(* Stop button *)
	xTmp:=	NOT(T_Visu.T_CtrleAction.xExecute);
	xTmpTeach:=((T_Visu.T_PlcParam.dwActualPage = 310) OR (T_Visu.T_PlcParam.dwActualPage = 410)) AND (bButtonPanelLocked = 16#10);
	IF xTmp THEN
		RisingEdgeStopButton(CLK:=xStopButton);
		IF RisingEdgeStopButton.Q AND ((bButtonPanelLocked = 16#0) OR xTmpTeach) THEN
		(* pane locked *)
			bButtonPanelLocked:=16#20;
			(* activ stop process *)
			T_Visu.T_CtrleAction.xExecute:=TRUE;
			CASE T_Visu.T_PlcParam.dwActualPage OF
			10:	T_Visu.T_CtrleAction.iFunction:=800;
			20:	T_Visu.T_CtrleAction.iFunction:=800;
			30:	T_Visu.T_CtrleAction.iFunction:=800;
			110:	T_Visu.T_CtrleAction.iFunction:=800;
				T_Visu.ptrT_ExchgParam^.T_Visu.T_Message.iState:=121;
			210:	T_Visu.T_CtrleAction.iFunction:=301;
				T_Visu.ptrT_ExchgParam^.T_Visu.T_Message.iState:=121;
			220:	T_Visu.T_CtrleAction.iFunction:=403;
				T_Visu.ptrT_ExchgParam^.T_Visu.T_Message.iState:=121;
			310:	T_Visu.T_CtrleAction.iFunction:=301;
				T_Visu.ptrT_ExchgParam^.T_Visu.T_Message.iState:=121;
			330:	T_Visu.T_CtrleAction.iFunction:=800;
				T_Visu.ptrT_ExchgParam^.T_Visu.T_Message.iState:=121;
			410:	T_Visu.T_CtrleAction.iFunction:=301;
				T_Visu.ptrT_ExchgParam^.T_Visu.T_Message.iState:=121;
			ELSE
				T_Visu.T_CtrleAction.xExecute:=FALSE;
			END_CASE
		END_IF
		(* manage falling edge stop button *)
		FallingEdgeStopButton(CLK:=xStopButton AND T_ConfigPage.xMaskBtStop);
		IF FallingEdgeStopButton.Q AND (bButtonPanelLocked AND 16#20) = 16#20 THEN
			bButtonPanelLocked:=bButtonPanelLocked XOR 16#20; END_IF
	ELSE
		RisingEdgeStopButton(CLK:=FALSE);
		FallingEdgeStopButton(CLK:=TRUE);
	END_IF
END_ACTION
ACTION CtrlTaskBar:
(* Management Bt navigation panel *)
	RisingEdgeTouchScreenNavPanel(CLK:=	T_Visu.ptrT_ExchgParam^.T_TouchScreenNavPanel.wActivBt <> 0);
	FallingEdgeTouchScreenNavPanel(CLK:=T_Visu.ptrT_ExchgParam^.T_TouchScreenNavPanel.wActivBt <> 0);
	xTmp:=	NOT(xChangePage)
			AND T_Visu.T_CtrleAction.xDone
			AND NOT(T_Visu.T_CtrleAction.xExecute)
			AND NOT(T_StartUp.T_State.xBlockChangeMovementVisu)
			AND NOT(T_StartUp.T_State.xBlockVisuNavigation)
			AND ((T_Visu.ptrT_ExchgParam^. T_TouchScreenNavPanel.wNotMasktext AND T_Visu.ptrT_ExchgParam^.T_TouchScreenNavPanel.wActivBt) <> 0);
	IF xTmp THEN
		(* activ action of rising edge *)
		IF RisingEdgeTouchScreenNavPanel.Q THEN
			ii:=1;
			wTmp:=T_Visu.ptrT_ExchgParam^.T_TouchScreenNavPanel.wActivBt;
			WHILE wTmp <> 16#0 DO
				IF (wTmp AND 16#1) = 16#1 THEN EXIT; END_IF
				wTmp:=ROR(wTmp,1);
				ii:=ii+1;
			END_WHILE
			T_Visu.T_CtrleAction.iFunction:=T_ConfigPage.aiFTrigActionTouchScreenNavPanel[ii];
			CASE T_Visu.ptrT_ExchgParam^.T_Visu.bActivSpecialLayer OF
				0: 	wNormalLayerActivTask:=T_Visu.ptrT_ExchgParam^.T_TouchScreenNavPanel.wActivBt;
					wNormalLayerActivPage:=T_Visu.T_CtrleAction.iFunction - 10000;
					T_Visu.ptrT_ExchgParam^.T_TouchScreenNavPanel.wState:=wNormalLayerActivTask;
					wTmpNormalLayerActivTask:=ii;
				1:	wSpecialLayerGeneralActivTask:=T_Visu.ptrT_ExchgParam^.T_TouchScreenNavPanel.wActivBt;
					wSpecialLayerGeneralActivPage:=T_Visu.T_CtrleAction.iFunction - 10000;
					T_Visu.ptrT_ExchgParam^.T_TouchScreenNavPanel.wState:=wSpecialLayerGeneralActivTask;
					wTmpSpecialLayerGeneralActivTask:=ii;
				2:	wSpecialLayerToolRotActivTask:=T_Visu.ptrT_ExchgParam^.T_TouchScreenNavPanel.wActivBt;
					wSpecialLayerToolRotActivPage:=T_Visu.T_CtrleAction.iFunction - 10000;
					T_Visu.ptrT_ExchgParam^.T_TouchScreenNavPanel.wState:=wSpecialLayerToolRotActivTask;
					wTmpSpecialLayerToolRotActivTask:=ii;
				3:	wSpecialLayerWireFeedActivTask:=T_Visu.ptrT_ExchgParam^.T_TouchScreenNavPanel.wActivBt;
					wSpecialLayerWireFeedActivPage:=T_Visu.T_CtrleAction.iFunction - 10000;
					T_Visu.ptrT_ExchgParam^.T_TouchScreenNavPanel.wState:=wSpecialLayerWireFeedActivTask;
					wTmpSpecialLayerWireFeedActivTask:=ii;
				4:	wSpecialLayerGrindAxisActivTask:=T_Visu.ptrT_ExchgParam^.T_TouchScreenNavPanel.wActivBt;
					wSpecialLayerGrindAxisActivPage:=T_Visu.T_CtrleAction.iFunction - 10000;
					T_Visu.ptrT_ExchgParam^.T_TouchScreenNavPanel.wState:=wSpecialLayerGrindAxisActivTask;
					wTmpSpecialLayerGrindAxisActivTask:=ii;
			END_CASE;
			IF ((INT_TO_WORD(T_Visu.ptrT_ExchgParam^.T_TouchScreenBtPanel.iStateBtLeft) AND 16#10) = 16#10) THEN
				T_Visu.T_CtrleAction.iFunction:=3;
				xResetParaListValue:=TRUE;
			END_IF;
			T_Visu.ptrT_ExchgParam^.T_TouchScreenNavPanel.wActivBt:=0;
			T_Visu.T_CtrleAction.xExecute:=TRUE;
		END_IF;
	ELSE
		T_Visu.ptrT_ExchgParam^.T_TouchScreenNavPanel.wActivBt:=0;
	END_IF;
(*22.12.2009: KFS 	{	*)
(* Management BT Tool  (additionel external buttons) only for MicroRod *)
	IF xMicroRodActive THEN
		(* ToolTension button *)
		xTmp:=	NOT(xChangePage) AND T_Visu.T_CtrleAction.xDone AND
				NOT(T_Visu.T_CtrleAction.xExecute) 	AND T_Visu.T_CtrleProcess.xDone AND (bStateMachine <>2);
		IF xTmp THEN
(*03.03.2017: KFS { *)
			RisingEdgeBtToolTension(CLK:=xToolTensionButton);
			IF RisingEdgeBtToolTension.Q THEN
				IF  T_Visu.ptrT_ExchgParam^.T_Cylinder.xToolTension AND	T_Visu.ptrT_ExchgParam^.T_Cylinder.xCylToolLeft AND T_Visu.ptrT_ExchgParam^.T_Cylinder.xCylToolRight	THEN
					T_Visu.T_CtrleAction.iFunction:=510;
					T_Visu.T_CtrleAction.xExecute:=TRUE;
				END_IF;
				IF  NOT (T_Visu.ptrT_ExchgParam^.T_Cylinder.xToolTension) THEN
					T_Visu.T_CtrleAction.iFunction:=510;
					T_Visu.T_CtrleAction.xExecute:=TRUE;
				END_IF;
			END_IF;
			RisingEdgeBtToolLeft(CLK:=xToolLeftButton);
			IF RisingEdgeBtToolLeft.Q THEN
				IF NOT T_Visu.ptrT_ExchgParam^.T_Cylinder.xToolTension  THEN
					T_Visu.T_CtrleAction.iFunction:=511;
					T_Visu.T_CtrleAction.xExecute:=TRUE;
				END_IF;
				IF  T_Visu.ptrT_ExchgParam^.T_Cylinder.xToolTension  AND NOT(T_Visu.ptrT_ExchgParam^.T_Cylinder.xCylToolLeft) THEN
					T_Visu.T_CtrleAction.iFunction:=511;
					T_Visu.T_CtrleAction.xExecute:=TRUE;
				END_IF;
			END_IF;
			RisingEdgeBtToolRight(CLK:=xToolRightButton);
			IF RisingEdgeBtToolRight.Q THEN
				IF NOT T_Visu.ptrT_ExchgParam^.T_Cylinder.xToolTension  THEN
					T_Visu.T_CtrleAction.iFunction:=512;
					T_Visu.T_CtrleAction.xExecute:=TRUE;
				END_IF;
				IF  T_Visu.ptrT_ExchgParam^.T_Cylinder.xToolTension  AND NOT(T_Visu.ptrT_ExchgParam^.T_Cylinder.xCylToolRight) THEN
					T_Visu.T_CtrleAction.iFunction:=512;
					T_Visu.T_CtrleAction.xExecute:=TRUE;
				END_IF;
			END_IF;
(*03.03.2017: KFS } *)
			RisingEdgeBtToolCenter(CLK:=xToolCenterButton);
			IF RisingEdgeBtToolCenter.Q THEN
				T_Visu.T_CtrleAction.iFunction:=513;
				T_Visu.T_CtrleAction.xExecute:=TRUE;
			END_IF;
			RisingEdgeBtToolPrismaLeft(CLK:=xToolPrismaLeftButton);
			IF RisingEdgeBtToolPrismaLeft.Q THEN
				T_Visu.T_CtrleAction.iFunction:=514;
				T_Visu.T_CtrleAction.xExecute:=TRUE;
			END_IF;
			RisingEdgeBtToolPrismaRight(CLK:=xToolPrismaRightButton);
			IF RisingEdgeBtToolPrismaRight.Q THEN
				T_Visu.T_CtrleAction.iFunction:=515;
				T_Visu.T_CtrleAction.xExecute:=TRUE;
			END_IF;
		ELSE
			IF   NOT(T_Visu.T_CtrleAction.xExecute) AND T_Visu.T_CtrleAction.xDone  THEN
				RisingEdgeBtToolTension(CLK:=FALSE);
				RisingEdgeBtToolLeft(CLK:=FALSE);
				RisingEdgeBtToolRight(CLK:=FALSE);
				RisingEdgeBtToolCenter(CLK:=FALSE);
				RisingEdgeBtToolPrismaLeft(CLK:=FALSE);
				RisingEdgeBtToolPrismaRight(CLK:=FALSE);
			END_IF;
		END_IF;
	END_IF;
(*22.12.2009: KFS 	}	*)
END_ACTION
ACTION CtrlVisuFunction:
(************************************************************************************************************************************************************************)
(***************                                          start of the management for call a function of the visualisation interface                                           ********************)
(************************************************************************************************************************************************************************)
(* waiting for executing action *)
	(* ...monitor Key panel "Enter" *)
	RisingEdgeKeyPanel_Enter(CLK:=T_Visu.ptrT_ExchgParam^.T_Visu.xKey_Enter);
	(* ...monitor Key panel "Esc" *)
	RisingEdgeKeyPanel_Esc(CLK:=T_Visu.ptrT_ExchgParam^.T_Visu.xKey_Escape);
	IF RisingEdgeKeyPanel_Esc.Q THEN tTimeOutAction:=TimerAction.ET; END_IF
	(*... not ready *)
	TimerNotReady(IN:=FALSE, PT:=T#2s);
	T_Visu.T_CtrleAction.xNotReady:=TimerNotReady.Q;

(* ...message *)
	RisingEdgeActionNotReady(CLK:=T_Visu.T_CtrleAction.xNotReady);
	IF RisingEdgeActionNotReady.Q AND T_Visu.ptrT_ExchgParam^.T_Visu.T_Message.iState < 200 THEN
		T_Visu.ptrT_ExchgParam^.T_Visu.T_Message.iState:=101; END_IF
	(* Release 'Not ready' action control structure *)
	FallingEdgeActionNotReady(CLK:=T_Visu.T_CtrleAction.xNotReady);
	IF FallingEdgeActionNotReady.Q THEN
		IF (T_Visu.ptrT_ExchgParam^.T_Visu.T_Message.iState =101) THEN
			T_Visu.ptrT_ExchgParam^.T_Visu.T_Message.iState:=0;
		END_IF;
		T_Visu.T_CtrleAction.xExecute:=FALSE;
		T_Visu.T_CtrleAction.xDone:=TRUE;
		T_Visu.T_CtrleAction.xErr:=FALSE;
		T_Visu.T_CtrleAction.udiErrorID:=0;
		iStepAction:=1;
		(*
		iStepActionRef:=1;
		iStepActionNovRam:=1;
		*)
		xStepActionDone:=FALSE;
		TimerAction(IN:=FALSE);
	END_IF
	(* ...done *)
	RisingEdgeActionDone(CLK:=T_Visu.T_CtrleAction.xDone);
	IF RisingEdgeActionDone.Q THEN
		(* disable mask stop action *)
		(*wStopActionMaskBtPanelRight:=16#0;*)
		(*xWaitingReleaseStopBtPanel:=FALSE;*)
		IF T_Visu.T_CtrleAction.iFunction > 100
		    AND (T_Visu.ptrT_ExchgParam^.T_Visu.T_Message.iState = 0 OR (T_Visu.ptrT_ExchgParam^.T_Visu.T_Message.iState  > 100 AND T_Visu.ptrT_ExchgParam^.T_Visu.T_Message.iState < 200)) THEN
			IF NOT TimerAction.Q AND NOT FallingEdgeActionNotReady.Q THEN
				IF NOT(xBlockConfirmMessage) THEN
					(* call confirmation message *)
					T_Visu.ptrT_ExchgParam^.T_Visu.T_Message.iState
						:=iFctReturnConfMessage(iNumAction:=T_Visu.T_CtrleAction.iFunction);
				ELSE
					xBlockConfirmMessage:=FALSE;
				END_IF;
			(* call cancelled message *)
			ELSE T_Visu.ptrT_ExchgParam^.T_Visu.T_Message.iState:=5; END_IF
		END_IF
	END_IF
	(* ...error *)
	RisingEdgeActionError(CLK:=T_Visu.T_CtrleAction.xErr);
	IF RisingEdgeActionError.Q THEN
	(* call function bloc action error *)
		(*fbQvisError(	udiActionError:=T_Visu.T_CtrleAction.udiErrorID,
					T_Message:=T_Visu.ptrT_ExchgParam^.T_Visu.T_Message);*)
		(* Init. variable *)
		T_Visu.T_CtrleAction.xExecute:=FALSE;
		T_Visu.T_CtrleAction.xDone:=TRUE;
		T_Visu.T_CtrleAction.xErr:=FALSE;
		T_Visu.T_CtrleAction.xNotReady:=FALSE;
		T_Visu.T_CtrleAction.udiErrorID:=0;
		iStepAction:=1;
		(*
		iStepActionRef:=1;
		iStepActionNovRam:=1;
		*)
		xStepActionDone:=FALSE;
	END_IF
	(* ...reset *)
	RisingEdgeResetAction(CLK:=T_Visu.T_CtrleAction.xReset);
	IF RisingEdgeResetAction.Q THEN
		(* Init. variable *)
		T_Visu.T_CtrleAction.xExecute:=FALSE;
		T_Visu.T_CtrleAction.xDone:=TRUE;
		T_Visu.T_CtrleAction.xErr:=FALSE;
		T_Visu.T_CtrleAction.xNotReady:=FALSE;
		T_Visu.T_CtrleAction.udiErrorID:=0;
		iStepAction:=1;
		(*
		iStepActionRef:=1;
		iStepActionNovRam:=1;
		*)
		xStepActionDone:=FALSE;
		TimerAction(IN:=FALSE);
		(* Release reset *)
		T_Visu.T_CtrleAction.xReset:=FALSE;
	END_IF

	(* Execute Function *)
	RisingEdgeExecuteAction(CLK:=T_Visu.T_CtrleAction.xExecute);
	IF RisingEdgeExecuteAction.Q THEN
		(* confirm action execution *)
		T_Visu.T_CtrleAction.xExecute:=FALSE;
		CASE T_Visu.T_CtrleAction.iFunction OF
			(* Set parameter page *)
			3:	xSetParameterPage:=TRUE;
				tTimeOutAction:=T#3s;
			(* Change Page Button Panel Left *)
			6:	xBtPanelLeftChangePage:=TRUE;
				tTimeOutAction:=T#3s;
	(*SOA 13.01.2023  { *)
			(* Change Page Button Panel Right *)
			7:	xBtPanelRightChangePage:=TRUE;
				tTimeOutAction:=T#3s;
	(*SOA 13.01.2023  } *)
			(* next page vertical *)
			12:	xNextPageVertical:=TRUE;
				tTimeOutAction:=T#3s;
			(* Delete error List *)
			20:	xDeleteErrorList:=TRUE;
				tTimeOutAction:=T#3s;
			(* Reset error *)
			99:	xResetError:=TRUE;
				tTimeOutAction:=T#3s;
			(* Open Overlay for input measured tool diameter *)
			101:	xOverlayMeasureToolDia:=TRUE;
				tTimeOutAction:=T#9999s;
			(* Plunge On/Off *)
			102:	xPlungeActivation:=TRUE;
				tTimeOutAction:=T#3s;
			(* Displace On/Off *)
			103:	xDisplaceActivation:=TRUE;
				tTimeOutAction:=T#3s;
			(* AutoGroove-->Block GrindFeeder On/Off *)
			104:	xBlockGrindFeederActivation:=TRUE;
				tTimeOutAction:=T#3s;
			(* AutoGroove-->ToolFeeder move to StartPos *)
			105:	xToolFeederMoveStartPos:=TRUE;
				tTimeOutAction:=T#3s;
			(* AutoGeometry and AutoGroove-->Switch On/Off all Axis Power *)
			106:	xToggleAllAxisPower:=TRUE;
				tTimeOutAction:=T#3s;
			(* AutoGeometry and AutoGroove-->ToolFeeder move to LoadPos *)
			107:	xToolFeederMoveLoadPos:=TRUE;
				tTimeOutAction:=T#3s;
(*08.07.2014: KFS	{	*)
			(* AutoGeometry -->WarmUp On/OFF *)
			108:	xWarmUp:=TRUE;
				tTimeOutAction:=T#3s;
(*08.07.2014: KFS	}	*)
			(* Correction Tool Diameter + *)
			110:	xCorrectionToolDiameterAdd:=TRUE;
				tTimeOutAction:=T#3s;
			(* Correction Tool Diameter ++ *)
			111:	xCorrectionToolDiameterAddMore:=TRUE;
				tTimeOutAction:=T#3s;
			(* Correction Tool Diameter - *)
			112:	xCorrectionToolDiameterSub:=TRUE;
				tTimeOutAction:=T#3s;
			(* Correction Tool Diameter -- *)
			113:	xCorrectionToolDiameterSubMore:=TRUE;
				tTimeOutAction:=T#3s;
			(* Reset Tool Diameter Correction *)
			114:	xResetToolDiameterCorrection:=TRUE;
				tTimeOutAction:=T#3s;
			(* Keypad Activation *)
			115: xKeyPadActivation:=TRUE;
				tTimeOutAction:=T#3s;
			(* Function Correction Tool Diameter *)
			116:	xFctCorrectionToolDiameter:=TRUE;
				tTimeOutAction:=T#3s;
			(* Select Prisma 1 or 2 Input *)
			120:	xSelectPrisma:=TRUE;
				tTimeOutAction:=T#3s;
			(* Set calculated ToolRotation Torque *)
			130:	xSetCalculToolRotTorque:=TRUE;
				tTimeOutAction:=T#3s;
			(* Reset calculated ToolRotation Torque *)
			131:	xResetCalculToolRotTorque:=TRUE;
				tTimeOutAction:=T#3s;
			(* Open Overlay for input the correction of the position of the GrindFeeder *)
			132:	xOverlayGrindFeedSetPlung:=TRUE;
				tTimeOutAction:=T#9999s;
	(*SOA 13.01.2023  { *)
			173:	xConfirmStartWarmUp:=TRUE;
				tTimeOutAction:=T#3s;
			(* Stop Warmupl  *)
			175: 	xStopWarmup:=TRUE;
				tTimeOutAction:=T#3s;
	(*SOA 13.01.2023  } *)
			(* Activation Section 1 *) (*
			201: (* 13.10.2010 KFS 	{ 	*)
				(*	xActivationSection1:=TRUE;
					tTimeOutAction:=T#3s;			*)
				(* 13.10.2010 KFS   }	 *) *)
			(* Activation Section 2 *)
			202:	xActivationSection2:=TRUE;
				tTimeOutAction:=T#3s;
			(* Activation Section 3 *)
			203:	xActivationSection3:=TRUE;
				tTimeOutAction:=T#3s;
			(* Activation Section 4 *)
			204:	xActivationSection4:=TRUE;
				tTimeOutAction:=T#3s;
			(* Set pitch equal *)
			205:	xSetPitchEqual:=TRUE;
				tTimeOutAction:=T#3s;
	(* 13.10.2022 SOA*)
			(* Activation Section 5 *)
			206:	xActivationSection5:=TRUE;
				tTimeOutAction:=T#3s;
			(* Activation Section 6 *)
			207:	xActivationSection6:=TRUE;
				tTimeOutAction:=T#3s;
	(* 13.10.2022 SOA*)
			(* TeachIN page *)
			301..399:	(* set pointer, default pointer axis slide *)
					ptrTeachINAxis:=ADR(T_Station.THardware.TAxisToolLeft);
					iSelectedAxis:=1;
					IF (T_Visu.T_PlcParam.dwActualPage = 210) THEN
						xSlowFast:=T_Visu.ptrT_ExchgParam^.T_TeachIn.xSlowFastToolRotation;
						CASE T_Visu.ptrT_ExchgParam^.T_TeachIn.iSelectAxisToolRotation OF
						1:	iSelectedAxis:=1;
							TParaAxisTeachIN:=T_Visu.ptrT_ExchgParam^.T_TeachIn.TParam_ToolLeft:=T_NovRam.T_Data.T_Standard.T_TeachINToolLeft;
							ptrTeachINAxis:=ADR(T_Station.THardware.TAxisToolLeft);
						2:	iSelectedAxis:=2;
							TParaAxisTeachIN:=T_Visu.ptrT_ExchgParam^.T_TeachIn.TParam_ToolCenter:=T_NovRam.T_Data.T_Standard.T_TeachINToolCenter;
							ptrTeachINAxis:=ADR(T_Station.THardware.TAxisToolCenter);
						3:	iSelectedAxis:=3;
							TParaAxisTeachIN:=T_Visu.ptrT_ExchgParam^.T_TeachIn.TParam_ToolRight:=T_NovRam.T_Data.T_Standard.T_TeachINToolRight;
							ptrTeachINAxis:=ADR(T_Station.THardware.TAxisToolRight);
						END_CASE
					END_IF;
					IF (T_Visu.T_PlcParam.dwActualPage = 30) OR (T_Visu.T_PlcParam.dwActualPage = 310) OR (T_Visu.T_PlcParam.dwActualPage = 320) OR (T_Visu.T_PlcParam.dwActualPage = 330) THEN
						iSelectedAxis:=4;
						xSlowFast:=T_Visu.ptrT_ExchgParam^.T_TeachIn.xSlowFastToolFeed;
						TParaAxisTeachIN:=T_Visu.ptrT_ExchgParam^.T_TeachIn.TParam_ToolFeeder:=T_NovRam.T_Data.T_Standard.T_TeachINToolFeeder;
						ptrTeachINAxis:=ADR(T_Station.THardware.TAxisToolFeeder);
					END_IF;
					IF (T_Visu.T_PlcParam.dwActualPage = 410) THEN
						xSlowFast:=T_Visu.ptrT_ExchgParam^.T_TeachIn.xSlowFastGrindFeeder;
						CASE T_Visu.ptrT_ExchgParam^.T_TeachIn.iSelectAxisGrind OF
						1:	iSelectedAxis:=5;
							TParaAxisTeachIN:=T_Visu.ptrT_ExchgParam^.T_TeachIn.TParam_GrindFeeder:=T_NovRam.T_Data.T_Standard.T_TeachINGrindFeeder;
							ptrTeachINAxis:=ADR(T_Station.THardware.TAxisGrindFeeder);
						2:	iSelectedAxis:=6;
							ptrTeachINAxis:=ADR(T_Station.THardware.TAxisGrindSpindle);
						END_CASE
					END_IF;
					CASE T_Visu.T_CtrleAction.iFunction OF
					(* Stop axis movement *)
					301:	xStopAxis:=TRUE;
						tTimeOutAction:=T#4s;
					(* Move Axis Absolut *)
					305:	IF (iSelectedAxis = 4) THEN
							IF xMicroRodActive THEN
								IF (T_Visu.ptrT_ExchgParam^.T_TeachIn.iSaveToolFeederPos = 0) THEN
									ptrTeachINAxis^.T_CtrleSingle.lrPosition:=T_Visu.ptrT_ExchgParam^.T_StationCommon.rNewToolFeederPosition;
								END_IF;
								IF (T_Visu.ptrT_ExchgParam^.T_TeachIn.iSaveToolFeederPos = 1) THEN
									ptrTeachINAxis^.T_CtrleSingle.lrPosition:=T_NovRam.T_Data.T_ProcessImageData.T_ProcessPara.rStartPosToolFeedAuto;
								END_IF;
								IF (T_Visu.ptrT_ExchgParam^.T_TeachIn.iSaveToolFeederPos = 2) THEN
									ptrTeachINAxis^.T_CtrleSingle.lrPosition:=T_NovRam.T_Data.T_ProcessImageData.T_CalibrationPara.rStartPosToolFeedCalib;
								END_IF;
								IF (T_Visu.ptrT_ExchgParam^.T_TeachIn.iSaveToolFeederPos = 3) THEN
									ptrTeachINAxis^.T_CtrleSingle.lrPosition:=T_NovRam.T_Data.T_ProcessImageData.T_CalibrationPara.rMeasurePosToolFeedCalib;
								END_IF;
								IF (T_Visu.ptrT_ExchgParam^.T_TeachIn.iSaveToolFeederPos = 4) THEN
									ptrTeachINAxis^.T_CtrleSingle.lrPosition:=T_NovRam.T_Data.T_Standard.T_AxisPosition.rLoadPosToolFeedAuto;
								END_IF;
								ptrTeachINAxis^.T_CtrleSingle.lrVelocity:=TParaAxisTeachIN.rPositionSpeed;
								xMoveAbsPosition:=TRUE;
							END_IF;
							IF NOT(xMicroRodActive) THEN
								ptrTeachINAxis^.T_CtrleSingle.lrDistance:=T_Visu.ptrT_ExchgParam^.T_StationCommon.rNewToolFeederPosition;
								ptrTeachINAxis^.T_CtrleSingle.lrVelocity:=TParaAxisTeachIN.rPositionSpeed;
								xMoveRelPosition:=TRUE;
							END_IF;
						END_IF;
						IF (iSelectedAxis = 5) THEN
							IF (T_Visu.ptrT_ExchgParam^.T_TeachIn.iSaveGrindFeederPos = 0) THEN
								ptrTeachINAxis^.T_CtrleSingle.lrPosition:=T_Visu.ptrT_ExchgParam^.T_StationCommon.rNewGrindFeederPosition;
							END_IF;
							IF (T_Visu.ptrT_ExchgParam^.T_TeachIn.iSaveGrindFeederPos = 1) THEN
								ptrTeachINAxis^.T_CtrleSingle.lrPosition:=T_NovRam.T_Data.T_ProcessImageData.T_ProcessPara.rToolDiameterProcess;
							END_IF;
							IF (T_Visu.ptrT_ExchgParam^.T_TeachIn.iSaveGrindFeederPos = 2) THEN
								ptrTeachINAxis^.T_CtrleSingle.lrPosition:=	T_NovRam.T_Data.T_ProcessImageData.T_ProcessPara.rToolDiameterProcess +
																	T_NovRam.T_Data.T_ProcessImageData.T_ProcessPara.rSecurityPosGrindFeedProcess;
							END_IF;
							IF (T_Visu.ptrT_ExchgParam^.T_TeachIn.iSaveGrindFeederPos = 3) THEN
								ptrTeachINAxis^.T_CtrleSingle.lrPosition:=T_NovRam.T_Data.T_ProcessImageData.T_PrismPara.rToolDiameterMin;;
							END_IF;
							IF (T_Visu.ptrT_ExchgParam^.T_TeachIn.iSaveGrindFeederPos = 4) THEN
								ptrTeachINAxis^.T_CtrleSingle.lrPosition:=T_NovRam.T_Data.T_ProcessImageData.T_PrismPara.rToolDiameterMax + T_NovRam.T_Data.T_Standard.T_TeachINGrindFeeder.rOffsetSWPosEndSwitch;
							END_IF;
							ptrTeachINAxis^.T_CtrleSingle.lrVelocity:=TParaAxisTeachIN.rPositionSpeed;
							xMoveAbsPosition:=TRUE;
						END_IF;
						tTimeOutAction:=T#999s;
					(* Move Inc Slow/Fast Pos *)
					310..311: IF NOT(xSlowFast) THEN
								ptrTeachINAxis^.T_CtrleSingle.lrDistance:=TParaAxisTeachIN.rIncSlow;
								ptrTeachINAxis^.T_CtrleSingle.lrVelocity:=TParaAxisTeachIN.rVelSlow;
							ELSE
								ptrTeachINAxis^.T_CtrleSingle.lrDistance:=TParaAxisTeachIN.rIncFast;
								ptrTeachINAxis^.T_CtrleSingle.lrVelocity:=TParaAxisTeachIN.rVelFast;
							END_IF
							xMoveRelPosition:=TRUE;
							tTimeOutAction:=T#200s;
					(* Move Inc Slow/Fast Neg *)
					312..313:	IF NOT(xSlowFast) THEN
								ptrTeachINAxis^.T_CtrleSingle.lrDistance:=TParaAxisTeachIN.rIncSlow * -1.0;
								ptrTeachINAxis^.T_CtrleSingle.lrVelocity:=TParaAxisTeachIN.rVelSlow;
							ELSE
								ptrTeachINAxis^.T_CtrleSingle.lrDistance:=TParaAxisTeachIN.rIncFast * -1.0;
								ptrTeachINAxis^.T_CtrleSingle.lrVelocity:=TParaAxisTeachIN.rVelFast;
							END_IF
							xMoveRelPosition:=TRUE;
							tTimeOutAction:=T#200s;
					(* Move Vel Slow/Fast Pos *)
					314..315:	IF NOT(xSlowFast) THEN
								ptrTeachINAxis^.T_CtrleSingle.lrVelocity:=TParaAxisTeachIN.rVelSlow;
							ELSE
								ptrTeachINAxis^.T_CtrleSingle.lrVelocity:=TParaAxisTeachIN.rVelFast;
							END_IF
							xMoveContinousVel:=TRUE;
							tTimeOutAction:=T#200s;
					(* Move Vel Slow/Fast Neg *)
					316..317:	IF NOT(xSlowFast) THEN
								ptrTeachINAxis^.T_CtrleSingle.lrVelocity:=TParaAxisTeachIN.rVelSlow * -1.0;
							ELSE
								ptrTeachINAxis^.T_CtrleSingle.lrVelocity:=TParaAxisTeachIN.rVelFast * -1.0;
							END_IF
							xMoveContinousVel:=TRUE;
							tTimeOutAction:=T#200s;
					(* Move Continuos Velocity *)
					318:		CASE iSelectedAxis OF
							1,2,3:	ptrTeachINAxis^.T_CtrleSingle.lrVelocity:=T_Visu.ptrT_ExchgParam^.T_StationCommon.rNewToolRotationSpeed;
							6:		ptrTeachINAxis^.T_CtrleSingle.lrVelocity:=T_Visu.ptrT_ExchgParam^.T_StationCommon.rNewGrindSpindleSpeed;
							END_CASE
							xMoveContinousVel:=TRUE;
							tTimeOutAction:=T#200s;
					(* Switch WireFeed Jog Speed Slow/Fast *)
					320:		IF ((iSelectedAxis = 1) OR (iSelectedAxis = 2) OR (iSelectedAxis = 3)) AND (T_Visu.T_PlcParam.dwActualPage <> 30) THEN
								xSlowFastJogToolRotation:=TRUE;
							END_IF;
							IF (iSelectedAxis = 4) OR (T_Visu.T_PlcParam.dwActualPage = 30) THEN
								xSlowFastJogToolFeeder:=TRUE;
							END_IF;
							IF (iSelectedAxis = 5) AND (T_Visu.T_PlcParam.dwActualPage <> 30) THEN
								xSlowFastJogGrindFeeder:=TRUE;
							END_IF;
							tTimeOutAction:=T#3s;
					(* Switch ToolRotation Master Slave *)
					321:		IF xMicroRodActive THEN
								(* ToolCenter --> Slave of ToolLeft only by MicroRod *)
								T_Station.THardware.TAxisToolCenter.T_CtrleSingle.lrGearDivider:=INT_TO_LREAL(T_Station.T_WorkTool.iBaseGearDivider);
								T_Station.THardware.TAxisToolCenter.T_CtrleSingle.lrGearFactor:=(	INT_TO_LREAL(T_Station.T_WorkTool.iBaseGearDivider) /
																								(T_Station.THardware.TAxisToolLeft.T_CtrleSingle.lrGearRatio /
																								T_Station.THardware.TAxisToolCenter.T_CtrleSingle.lrGearRatio)) * -1.0;

								(* ToolRight --> Slave of ToolLeft by MicroWire or Slave of ToolRight by MicroRod *)
								T_Station.THardware.TAxisToolRight.T_CtrleSingle.lrGearDivider:=INT_TO_LREAL(T_Station.T_WorkTool.iBaseGearDivider);
								T_Station.THardware.TAxisToolRight.T_CtrleSingle.lrGearFactor:=	INT_TO_LREAL(T_Station.T_WorkTool.iBaseGearDivider) /
																								(T_Station.THardware.TAxisToolLeft.T_CtrleSingle.lrGearRatio /
																								T_Station.THardware.TAxisToolRight.T_CtrleSingle.lrGearRatio);
							END_IF;
							IF NOT(xMicroRodActive) THEN
								(* ToolRight --> Slave of ToolRight by MicroWire *)
								T_Station.THardware.TAxisToolFeeder.T_CtrleSingle.lrGearDivider:=INT_TO_LREAL(T_Station.T_WorkTool.iBaseGearDivider);
								T_Station.THardware.TAxisToolFeeder.T_CtrleSingle.lrGearFactor:=	(INT_TO_LREAL(T_Station.T_WorkTool.iBaseGearDivider) /
																							(T_Station.THardware.TAxisToolFeeder.T_CtrleSingle.lrGearRatio /
																							T_Station.THardware.TAxisToolRight.T_CtrleSingle.lrGearRatio)) * -1.0;

								(* ToolRight --> Slave of ToolLeft by MicroWire or Slave of ToolRight by MicroRod *)
								T_Station.THardware.TAxisToolRight.T_CtrleSingle.lrGearDivider:=INT_TO_LREAL(T_Station.T_WorkTool.iBaseGearDivider);
								T_Station.THardware.TAxisToolRight.T_CtrleSingle.lrGearFactor:=	(INT_TO_LREAL(T_Station.T_WorkTool.iBaseGearDivider) /
																								(T_Station.THardware.TAxisToolLeft.T_CtrleSingle.lrGearRatio /
																								T_Station.THardware.TAxisToolRight.T_CtrleSingle.lrGearRatio)) * -1.0;
							END_IF;
							xSwitchMasterSlave:=TRUE;
							tTimeOutAction:=T#3s;
					(* Power axis *)
					322:		xToggleAxisPower:=TRUE;
							tTimeOutAction:=T#3s;
					(* Reset axis *)
					323:		xResetAxis:=TRUE;
							tTimeOutAction:=T#3s;
					(* Reference axis *)
					324:		xReferenceAxis:=TRUE;
							tTimeOutAction:=T#200s;
					(* Teach axis Position *)
					325:		xTeachPosition:=TRUE;
							tTimeOutAction:=T#6s;
					(* Calculate the position between the RefIndex and the RefSensor *)
					326:		xCalcAngleRefIndex:=TRUE;
							tTimeOutAction:=T#200s;

					(* CW /CCW *)
					330:		xCWCCW:=TRUE;
							tTimeOutAction:=T#3s;
					(* CylBrake *)
					331:		xCylBrake:=TRUE;
							tTimeOutAction:=T#3s;
					END_CASE;
			(* Station Function *)
			401..499:	xActivateStationFunction:=TRUE;
					iTmpStationFunctionNr:=T_Visu.T_CtrleAction.iFunction - 400;	(* Select Function Number 1 - 99 *)
					IF (iTmpStationFunctionNr = 20) THEN tTimeOutAction:=T#200s; ELSE tTimeOutAction:=T#3s;END_IF;
			(* Cylinder Function *)
			501..599:	(* set pointer, default pointer CylToolTension *)
					(* 1=CylToolTension, 2=CylToolLeftActive, 3=CylToolRightActive, 4=CylToolCenter,5=CylToolPrismaLeftActive, 6=CylToolPrismaRightActive *)
					ptrCylAction:=ADR(T_Station.THardware.TCylToolTension);
					iSelectedCylinder:=1;
					IF (T_Visu.T_PlcParam.dwActualPage = 230) THEN
						IF (T_Visu.ptrT_ExchgParam^.T_Cylinder.iSelectCylinder_Sonder1 = 1) THEN
							ptrCylAction:=ADR(T_Station.THardware.TCylToolTension);
							iSelectedCylinder:=1;
						ELSIF (T_Visu.ptrT_ExchgParam^.T_Cylinder.iSelectCylinder_Sonder1 = 2) THEN
							ptrCylAction:=ADR(T_Station.THardware.TCylToolLeftActive);
							iSelectedCylinder:=2;
						ELSIF (T_Visu.ptrT_ExchgParam^.T_Cylinder.iSelectCylinder_Sonder1 = 3) THEN
							ptrCylAction:=ADR(T_Station.THardware.TCylToolRightActive);
							iSelectedCylinder:=3;
						ELSIF (T_Visu.ptrT_ExchgParam^.T_Cylinder.iSelectCylinder_Sonder1 = 4) THEN
							ptrCylAction:=ADR(T_Station.THardware.TCylToolCenterActive);
							iSelectedCylinder:=4;
						ELSIF (T_Visu.ptrT_ExchgParam^.T_Cylinder.iSelectCylinder_Sonder1 = 5) THEN
							ptrCylAction:=ADR(T_Station.THardware.TCylToolPrismaLeftActive);
							iSelectedCylinder:=5;
						ELSIF (T_Visu.ptrT_ExchgParam^.T_Cylinder.iSelectCylinder_Sonder1 = 6) THEN
							ptrCylAction:=ADR(T_Station.THardware.TCylToolPrismaRightActive);
							iSelectedCylinder:=6;
						ELSE
							ptrCylAction:=ADR(T_Station.THardware.TCylToolTension);
							iSelectedCylinder:=1;
						END_IF;
					END_IF;
					(*Set pointer -->selection by the extern buttons*)
					IF (T_Visu.T_CtrleAction.iFunction = 510) THEN ptrCylAction:=ADR(T_Station.THardware.TCylToolTension);iSelectedCylinder:=1; END_IF;
					IF (T_Visu.T_CtrleAction.iFunction = 511) THEN ptrCylAction:=ADR(T_Station.THardware.TCylToolLeftActive);iSelectedCylinder:=2; END_IF;
					IF (T_Visu.T_CtrleAction.iFunction = 512) THEN ptrCylAction:=ADR(T_Station.THardware.TCylToolRightActive);iSelectedCylinder:=3; END_IF;
					IF (T_Visu.T_CtrleAction.iFunction = 513) THEN ptrCylAction:=ADR(T_Station.THardware.TCylToolCenterActive);iSelectedCylinder:=4; END_IF;
					IF (T_Visu.T_CtrleAction.iFunction = 514) THEN ptrCylAction:=ADR(T_Station.THardware.TCylToolPrismaLeftActive);iSelectedCylinder:=5; END_IF;
					IF (T_Visu.T_CtrleAction.iFunction = 515) THEN ptrCylAction:=ADR(T_Station.THardware.TCylToolPrismaRightActive);iSelectedCylinder:=6; END_IF;
					IF ((T_Visu.T_CtrleAction.iFunction >= 510) AND (T_Visu.T_CtrleAction.iFunction <= 515)) THEN
						T_Visu.T_CtrleAction.iFunction:=501;
					 END_IF;
					CASE T_Visu.T_CtrleAction.iFunction OF
					501:		xToggleCylinderState:=TRUE;
							IF ( iSelectedCylinder = 1) THEN
								IF (T_Visu.T_PlcParam.dwActualPage = 220) THEN
									ptrCylAction^.T_CtrleCyl.T_AnalogCylinder.rForceIn:=T_Visu.ptrT_ExchgParam^.T_InfoValueCommon.rToolTensionForce;
								ELSE
									IF (T_Visu.ptrT_ExchgParam^.T_Cylinder.iSelectToolTensionForce < 2) THEN
										(* Process work force *)
										ptrCylAction^.T_CtrleCyl.T_AnalogCylinder.rForceIn:=T_NovRam.T_Data.T_ProcessImageData.T_ProcessPara.rToolTensionProcess;
									END_IF;
									IF (T_Visu.ptrT_ExchgParam^.T_Cylinder.iSelectToolTensionForce > 1) THEN
										(* Setup (Cylinder Force) Force *)
										ptrCylAction^.T_CtrleCyl.T_AnalogCylinder.rForceIn:=T_NovRam.T_Data.T_Standard.T_Cyl_ToolTension.rForce;
									END_IF;
								END_IF;
							END_IF;
							tTimeOutAction:=T#2s;
					(* ToolTens force + *)
					502:		xToolTensForceAdd:=TRUE;
							tTimeOutAction:=T#2s;
					(* ToolTens force ++ *)
					503:		xToolTensForceAddMore:=TRUE;
							tTimeOutAction:=T#2s;
					(* ToolTens force - *)
					504:		xToolTensForceSub:=TRUE;
							tTimeOutAction:=T#2s;
					(* ToolTens force -- *)
					505:		xToolTensForceSubMore:=TRUE;
							tTimeOutAction:=T#2s;
					(* DO NOT USE FUNCTION 510,511,512,513,514,515 *)
					END_CASE;
			(* All process station *)
			601..699:	T_Process.iFunctNr:=T_Visu.T_CtrleAction.iFunction - 600;
					xActionProcStation:=TRUE;
					tTimeOutAction:=T#2s;
			(* All process machine *)
			701..799:	T_Process.iFunctNr:=T_Visu.T_CtrleAction.iFunction - 700;
					xActionProcMachine:=TRUE;
					(* Ref timeout 120s *)
					IF T_Visu.T_CtrleAction.iFunction = 710 THEN  tTimeOutAction:=T#120s; ELSE tTimeOutAction:=T#0.5s; END_IF
			(* Stop process *)
			800:		xStopProcess:=TRUE;
					tTimeOutAction:=T#30s;
			(* Stop cycle *)
			801:		xAction_StopCycle:=TRUE;
					tTimeOutAction:=T#30s;
			(* Copy profile to process value *)
			1001:	xAction_CopyProfileToProcess:=TRUE;
					tTimeOutAction:=T#10s;
			(* Load profile to process image *)
			1002:	xAction_LoadProfileToProcessImage:=TRUE;
					tTimeOutAction:=T#5s;
			(* Save profile to File *)
			1003:	xAction_SaveProfileToFile:=TRUE;
					tTimeOutAction:=T#5s;
			(* Delete Profile *)
			1004:	xActionDeleteProfile:=TRUE;
					tTimeOutAction:=T#5s;
			(* Save NovRAM with confirmation *)
			1005:	xAction_SaveNovRAM:=TRUE;
					tTimeOutAction:=T#6s;
			(* Save NovRAM without confirmation *)
			1006:	xAction_SaveNovRAMWithoutConfirm:=TRUE;
					tTimeOutAction:=T#10s;
			(* change page *)
			10001..10999:	xNavPanelChangePage:=TRUE;
						tTimeOutAction:=T#3s;
		END_CASE;
		(* Init. variable *)
		T_Visu.T_CtrleAction.xDone:=FALSE;
		T_Visu.T_CtrleAction.xNotReady:=FALSE;
		T_Visu.T_CtrleAction.xErr:=FALSE;
		T_Visu.T_CtrleAction.udiErrorID:=0;
		iStepAction:=1;
		iStepActionNovRam:=1;
		xStepActionDone:=FALSE;
		IF tTimeOutAction <> T#0s THEN TimerAction(IN:=FALSE); END_IF
		(* exit FB *)
		RETURN;
	END_IF;

(* Timer action *)
	IF tTimeOutAction <> T#0s THEN TimerAction(IN:=TRUE,PT:=tTimeOutAction); END_IF
	RisingEdgeTimeOut(CLK:=TimerAction.Q);
	IF RisingEdgeTimeOut.Q AND NOT(T_Visu.T_CtrleAction.xDone) AND NOT(T_Visu.T_CtrleAction.xErr) THEN
	(* Timeout action activ *)
		T_Visu.T_CtrleAction.xExecute:=FALSE;
		T_Visu.T_CtrleAction.xDone:=TRUE;
		T_Visu.T_CtrleAction.xNotReady:=FALSE;
		T_Visu.T_CtrleAction.xErr:=FALSE;
		T_Visu.T_CtrleAction.udiErrorID:=16#0;
		(* call confirmation message *)
		T_Visu.ptrT_ExchgParam^.T_Visu.T_Message.iState:=102;
(*			:=iFctReturnConfMessage(iNumAction:=-1);*)
		(* exit FB, do not continue the execution of action! *)
		RETURN;
	END_IF
(************************************************************************************************************************************************************************)
(***************                                          end  of the management for call a function of the visualisation interface                                           ********************)
(************************************************************************************************************************************************************************)
END_ACTION
ACTION MaskFunctionButton:
CASE T_Visu.T_PlcParam.dwActualPage OF
410:	CASE T_Visu.ptrT_ExchgParam^.T_TeachIn.iSelectAxisGrind OF
	1:	wForceMaskFunctionPanel:=16#2B;
		aiForceRTrigActionFunctionPanel[1]:=322;		(* On/Off *)
		aiForceRTrigActionFunctionPanel[2]:=323;		(* Reset *)
		aiForceRTrigActionFunctionPanel[3]:=0;
		aiForceRTrigActionFunctionPanel[4]:=320;		(* Slow / Fast *)
		aiForceRTrigActionFunctionPanel[5]:=0;
		aiForceRTrigActionFunctionPanel[6]:=325;		(* Save position *)
	2:	wForceMaskFunctionPanel:=16#2B;
		aiForceRTrigActionFunctionPanel[1]:=322;		(* On/Off *)
		aiForceRTrigActionFunctionPanel[2]:=323;		(* Reset *)
		aiForceRTrigActionFunctionPanel[3]:=0;
		aiForceRTrigActionFunctionPanel[4]:=330;		(* CW / CCW *)
		aiForceRTrigActionFunctionPanel[5]:=0;
		aiForceRTrigActionFunctionPanel[6]:=331;		(* CylBrake *)
	END_CASE
END_CASE
END_ACTION
ACTION Monitor_ActuatorState:
(* Monitoring Axis value *)
	(* ToolLeft Monitoring *)
	IF T_Station.THardware.TAxisToolLeft.T_CtrleSingle.xPower THEN
		T_Visu.ptrT_ExchgParam^.T_StationCommon.bStateAxisReelLeft:=T_Visu.ptrT_ExchgParam^.T_StationCommon.bStateAxisReelLeft OR 16#1;
	ELSE
		T_Visu.ptrT_ExchgParam^.T_StationCommon.bStateAxisReelLeft:=T_Visu.ptrT_ExchgParam^.T_StationCommon.bStateAxisReelLeft AND 16#FE;
	END_IF;
	IF NOT(T_Station.THardware.TAxisToolLeft.T_CtrleSingle.xNotMoving) THEN
		T_Visu.ptrT_ExchgParam^.T_StationCommon.bStateAxisReelLeft:=T_Visu.ptrT_ExchgParam^.T_StationCommon.bStateAxisReelLeft OR 16#2;
	ELSE
		T_Visu.ptrT_ExchgParam^.T_StationCommon.bStateAxisReelLeft:=T_Visu.ptrT_ExchgParam^.T_StationCommon.bStateAxisReelLeft AND 16#FD;
	END_IF;
	IF T_Station.THardware.TAxisToolLeft.T_CtrleSingle.xErr THEN
		T_Visu.ptrT_ExchgParam^.T_StationCommon.bStateAxisReelLeft:=T_Visu.ptrT_ExchgParam^.T_StationCommon.bStateAxisReelLeft OR 16#4;
	ELSE
		T_Visu.ptrT_ExchgParam^.T_StationCommon.bStateAxisReelLeft:=T_Visu.ptrT_ExchgParam^.T_StationCommon.bStateAxisReelLeft AND 16#FB;
	END_IF;
	(* ToolRight Monitoring *)
	IF T_Station.THardware.TAxisToolRight.T_CtrleSingle.xPower THEN
		T_Visu.ptrT_ExchgParam^.T_StationCommon.bStateAxisReelRight:=T_Visu.ptrT_ExchgParam^.T_StationCommon.bStateAxisReelRight OR 16#1;
	ELSE
		T_Visu.ptrT_ExchgParam^.T_StationCommon.bStateAxisReelRight:=T_Visu.ptrT_ExchgParam^.T_StationCommon.bStateAxisReelRight AND 16#FE;
	END_IF;
	IF NOT(T_Station.THardware.TAxisToolRight.T_CtrleSingle.xNotMoving) THEN
		T_Visu.ptrT_ExchgParam^.T_StationCommon.bStateAxisReelRight:=T_Visu.ptrT_ExchgParam^.T_StationCommon.bStateAxisReelRight OR 16#2;
	ELSE
		T_Visu.ptrT_ExchgParam^.T_StationCommon.bStateAxisReelRight:=T_Visu.ptrT_ExchgParam^.T_StationCommon.bStateAxisReelRight AND 16#FD;
	END_IF;
	IF T_Station.THardware.TAxisToolRight.T_CtrleSingle.xErr THEN
		T_Visu.ptrT_ExchgParam^.T_StationCommon.bStateAxisReelRight:=T_Visu.ptrT_ExchgParam^.T_StationCommon.bStateAxisReelRight OR 16#4;
	ELSE
		T_Visu.ptrT_ExchgParam^.T_StationCommon.bStateAxisReelRight:=T_Visu.ptrT_ExchgParam^.T_StationCommon.bStateAxisReelRight AND 16#FB;
	END_IF;
	IF T_Station.THardware.TAxisToolRight.T_CtrleSingle.xSlave THEN
		T_Visu.ptrT_ExchgParam^.T_StationCommon.bStateAxisReelRight:=T_Visu.ptrT_ExchgParam^.T_StationCommon.bStateAxisReelRight OR 16#8;
	ELSE
		T_Visu.ptrT_ExchgParam^.T_StationCommon.bStateAxisReelRight:=T_Visu.ptrT_ExchgParam^.T_StationCommon.bStateAxisReelRight AND 16#F7;
	END_IF;
	(* ToolCenter Monitoring *)
	IF T_Station.THardware.TAxisToolCenter.T_CtrleSingle.xPower THEN
		T_Visu.ptrT_ExchgParam^.T_StationCommon.bStateAxisReelCenter:=T_Visu.ptrT_ExchgParam^.T_StationCommon.bStateAxisReelCenter OR 16#1;
	ELSE
		T_Visu.ptrT_ExchgParam^.T_StationCommon.bStateAxisReelCenter:=T_Visu.ptrT_ExchgParam^.T_StationCommon.bStateAxisReelCenter AND 16#FE;
	END_IF;
	IF NOT(T_Station.THardware.TAxisToolCenter.T_CtrleSingle.xNotMoving) THEN
		T_Visu.ptrT_ExchgParam^.T_StationCommon.bStateAxisReelCenter:=T_Visu.ptrT_ExchgParam^.T_StationCommon.bStateAxisReelCenter OR 16#2;
	ELSE
		T_Visu.ptrT_ExchgParam^.T_StationCommon.bStateAxisReelCenter:=T_Visu.ptrT_ExchgParam^.T_StationCommon.bStateAxisReelCenter AND 16#FD;
	END_IF;
	IF T_Station.THardware.TAxisToolCenter.T_CtrleSingle.xErr THEN
		T_Visu.ptrT_ExchgParam^.T_StationCommon.bStateAxisReelCenter:=T_Visu.ptrT_ExchgParam^.T_StationCommon.bStateAxisReelCenter OR 16#4;
	ELSE
		T_Visu.ptrT_ExchgParam^.T_StationCommon.bStateAxisReelCenter:=T_Visu.ptrT_ExchgParam^.T_StationCommon.bStateAxisReelCenter AND 16#FB;
	END_IF;
	IF T_Station.THardware.TAxisToolCenter.T_CtrleSingle.xSlave THEN
		T_Visu.ptrT_ExchgParam^.T_StationCommon.bStateAxisReelCenter:=T_Visu.ptrT_ExchgParam^.T_StationCommon.bStateAxisReelCenter OR 16#8;
	ELSE
		T_Visu.ptrT_ExchgParam^.T_StationCommon.bStateAxisReelCenter:=T_Visu.ptrT_ExchgParam^.T_StationCommon.bStateAxisReelCenter AND 16#F7;
	END_IF;
	(* ToolFeeder Monitoring *)
	IF T_Station.THardware.TAxisToolFeeder.T_CtrleSingle.xPower THEN
		T_Visu.ptrT_ExchgParam^.T_StationCommon.bStateAxisWireFeeder:=T_Visu.ptrT_ExchgParam^.T_StationCommon.bStateAxisWireFeeder OR 16#1;
	ELSE
		T_Visu.ptrT_ExchgParam^.T_StationCommon.bStateAxisWireFeeder:=T_Visu.ptrT_ExchgParam^.T_StationCommon.bStateAxisWireFeeder AND 16#FE;
	END_IF;
	IF NOT(T_Station.THardware.TAxisToolFeeder.T_CtrleSingle.xNotMoving) THEN
		T_Visu.ptrT_ExchgParam^.T_StationCommon.bStateAxisWireFeeder:=T_Visu.ptrT_ExchgParam^.T_StationCommon.bStateAxisWireFeeder OR 16#2;
	ELSE
		T_Visu.ptrT_ExchgParam^.T_StationCommon.bStateAxisWireFeeder:=T_Visu.ptrT_ExchgParam^.T_StationCommon.bStateAxisWireFeeder AND 16#FD;
	END_IF;
	IF T_Station.THardware.TAxisToolFeeder.T_CtrleSingle.xErr THEN
		T_Visu.ptrT_ExchgParam^.T_StationCommon.bStateAxisWireFeeder:=T_Visu.ptrT_ExchgParam^.T_StationCommon.bStateAxisWireFeeder OR 16#4;
	ELSE
		T_Visu.ptrT_ExchgParam^.T_StationCommon.bStateAxisWireFeeder:=T_Visu.ptrT_ExchgParam^.T_StationCommon.bStateAxisWireFeeder AND 16#FB;
	END_IF;
	IF T_Station.THardware.TAxisToolFeeder.T_CtrleSingle.xSlave THEN
		T_Visu.ptrT_ExchgParam^.T_StationCommon.bStateAxisWireFeeder:=T_Visu.ptrT_ExchgParam^.T_StationCommon.bStateAxisWireFeeder OR 16#8;
	ELSE
		T_Visu.ptrT_ExchgParam^.T_StationCommon.bStateAxisWireFeeder:=T_Visu.ptrT_ExchgParam^.T_StationCommon.bStateAxisWireFeeder AND 16#F7;
	END_IF;
	(* GrindFeeder Monitoring *)
	IF T_Station.THardware.TAxisGrindFeeder.T_CtrleSingle.xPower THEN
		T_Visu.ptrT_ExchgParam^.T_StationCommon.bStateAxisGrind:=T_Visu.ptrT_ExchgParam^.T_StationCommon.bStateAxisGrind OR 16#1;
	ELSE
		T_Visu.ptrT_ExchgParam^.T_StationCommon.bStateAxisGrind:=T_Visu.ptrT_ExchgParam^.T_StationCommon.bStateAxisGrind AND 16#FE;
	END_IF;
	IF NOT(T_Station.THardware.TAxisGrindFeeder.T_CtrleSingle.xNotMoving) THEN
		T_Visu.ptrT_ExchgParam^.T_StationCommon.bStateAxisGrind:=T_Visu.ptrT_ExchgParam^.T_StationCommon.bStateAxisGrind OR 16#2;
	ELSE
		T_Visu.ptrT_ExchgParam^.T_StationCommon.bStateAxisGrind:=T_Visu.ptrT_ExchgParam^.T_StationCommon.bStateAxisGrind AND 16#FD;
	END_IF;
	IF T_Station.THardware.TAxisGrindFeeder.T_CtrleSingle.xErr THEN
		T_Visu.ptrT_ExchgParam^.T_StationCommon.bStateAxisGrind:=T_Visu.ptrT_ExchgParam^.T_StationCommon.bStateAxisGrind OR 16#4;
	ELSE
		T_Visu.ptrT_ExchgParam^.T_StationCommon.bStateAxisGrind:=T_Visu.ptrT_ExchgParam^.T_StationCommon.bStateAxisGrind AND 16#FB;
	END_IF;
	IF T_Station.THardware.TAxisGrindFeeder.T_CtrleSingle.xSlave THEN
		T_Visu.ptrT_ExchgParam^.T_StationCommon.bStateAxisGrind:=T_Visu.ptrT_ExchgParam^.T_StationCommon.bStateAxisGrind OR 16#8;
	ELSE
		T_Visu.ptrT_ExchgParam^.T_StationCommon.bStateAxisGrind:=T_Visu.ptrT_ExchgParam^.T_StationCommon.bStateAxisGrind AND 16#F7;
	END_IF;
	(* GrindSpindle Monitoring *)
	IF T_Station.THardware.TAxisGrindSpindle.T_CtrleSingle.xPower THEN
		T_Visu.ptrT_ExchgParam^.T_StationCommon.bStateAxisGrindSpindle:=T_Visu.ptrT_ExchgParam^.T_StationCommon.bStateAxisGrindSpindle OR 16#1;
	ELSE
		T_Visu.ptrT_ExchgParam^.T_StationCommon.bStateAxisGrindSpindle:=T_Visu.ptrT_ExchgParam^.T_StationCommon.bStateAxisGrindSpindle AND 16#FE;
	END_IF;
	IF NOT(T_Station.THardware.TAxisGrindSpindle.T_CtrleSingle.xNotMoving) THEN
		T_Visu.ptrT_ExchgParam^.T_StationCommon.bStateAxisGrindSpindle:=T_Visu.ptrT_ExchgParam^.T_StationCommon.bStateAxisGrindSpindle OR 16#2;
	ELSE
		T_Visu.ptrT_ExchgParam^.T_StationCommon.bStateAxisGrindSpindle:=T_Visu.ptrT_ExchgParam^.T_StationCommon.bStateAxisGrindSpindle AND 16#FD;
	END_IF;
	IF T_Station.THardware.TAxisGrindSpindle.T_CtrleSingle.xErr THEN
		T_Visu.ptrT_ExchgParam^.T_StationCommon.bStateAxisGrindSpindle:=T_Visu.ptrT_ExchgParam^.T_StationCommon.bStateAxisGrindSpindle OR 16#4;
	ELSE
		T_Visu.ptrT_ExchgParam^.T_StationCommon.bStateAxisGrindSpindle:=T_Visu.ptrT_ExchgParam^.T_StationCommon.bStateAxisGrindSpindle AND 16#FB;
	END_IF;
	(* General Actual Axis value *)
	T_Visu.ptrT_ExchgParam^.T_InfoValueCommon.rActualToolRotSpeed:=T_Station.THardware.TAxisToolLeft.T_LiveValue.lrActualVelocity;
	IF (T_Visu.ptrT_ExchgParam^.T_TeachIn.iSelectAxisToolRotation = 1) THEN
		T_Visu.ptrT_ExchgParam^.T_StationCommon.rActualToolRotationSpeed:=T_Station.THardware.TAxisToolLeft.T_LiveValue.lrActualVelocity;
	END_IF;
	IF (T_Visu.ptrT_ExchgParam^.T_TeachIn.iSelectAxisToolRotation = 2) THEN
		T_Visu.ptrT_ExchgParam^.T_StationCommon.rActualToolRotationSpeed:=T_Station.THardware.TAxisToolCenter.T_LiveValue.lrActualVelocity;
	END_IF;
	IF (T_Visu.ptrT_ExchgParam^.T_TeachIn.iSelectAxisToolRotation = 3) THEN
		T_Visu.ptrT_ExchgParam^.T_StationCommon.rActualToolRotationSpeed:=T_Station.THardware.TAxisToolRight.T_LiveValue.lrActualVelocity;
	END_IF;
	IF xMicroRodActive THEN
		IF (T_Visu.T_PlcParam.dwActualPage = 10) OR (T_Visu.T_PlcParam.dwActualPage = 20) THEN
			T_Visu.ptrT_ExchgParam^.T_InfoValueCommon.rActualWireFeedPosition:=	T_Station.THardware.TAxisToolFeeder.T_LiveValue.lrActualPosition -
																						T_NovRam.T_Data.T_ProcessImageData.T_ProcessPara.rStartPosToolFeedAuto;
		END_IF;
		IF (T_Visu.T_PlcParam.dwActualPage = 110) THEN
			T_Visu.ptrT_ExchgParam^.T_InfoValueCommon.rActualWireFeedPosition:=	T_Station.THardware.TAxisToolFeeder.T_LiveValue.lrActualPosition -
																						T_NovRam.T_Data.T_ProcessImageData.T_CalibrationPara.rStartPosToolFeedCalib;
		END_IF;
		IF (T_Visu.T_PlcParam.dwActualPage = 30) THEN
			T_Visu.ptrT_ExchgParam^.T_InfoValueCommon.rActualWireFeedPosition:=	T_Station.THardware.TAxisToolFeeder.T_LiveValue.lrActualPosition;
		END_IF;
		IF (T_Visu.T_PlcParam.dwActualPage = 330) THEN
			T_Visu.ptrT_ExchgParam^.T_InfoValueCommon.rActualWireFeedPosition:=	T_Station.THardware.TAxisToolFeeder.T_LiveValue.lrActualPosition;
		END_IF;
		T_Visu.ptrT_ExchgParam^.T_StationCommon.rActualToolFeederPosition:=T_Station.THardware.TAxisToolFeeder.T_LiveValue.lrActualPosition;
		T_Visu.ptrT_ExchgParam^.T_InfoValueCommon.rActualWireFeedSpeed:=T_Station.THardware.TAxisToolFeeder.T_LiveValue.lrActualVelocity;
	ELSE
		(* On the MicroWire set the Position of the ToolFeed every time when the TeachPage will be activate to zero *)
		IF (T_Visu.T_PlcParam.dwActualPage = 310) AND NOT(xReadActualToolFeedPos) THEN
			rActualToolFeederPosition:=T_Station.THardware.TAxisToolFeeder.T_LiveValue.lrActualPosition;
			xReadActualToolFeedPos:=TRUE;
		END_IF;
		IF (T_Visu.T_PlcParam.dwActualPage <> 310) THEN
			xReadActualToolFeedPos:=FALSE;
		END_IF;
		T_Visu.ptrT_ExchgParam^.T_StationCommon.rActualToolFeederPosition:=T_Station.THardware.TAxisToolFeeder.T_LiveValue.lrActualPosition - rActualToolFeederPosition;
		(* On the MicroWire set the Position of the ToolFeed every time when the Reference Page will be activate to zero *)
		IF (T_Visu.T_PlcParam.dwActualPage = 30) AND NOT(xReadActualToolFeedPos1) THEN
			rActualToolFeederPosition1:=T_Station.THardware.TAxisToolFeeder.T_LiveValue.lrActualPosition;
			xReadActualToolFeedPos1:=TRUE;
		END_IF;
		IF (T_Visu.T_PlcParam.dwActualPage <> 30) THEN
			xReadActualToolFeedPos1:=FALSE;
		END_IF;
		IF (T_Visu.T_PlcParam.dwActualPage = 30) THEN
			T_Visu.ptrT_ExchgParam^.T_InfoValueCommon.rActualWireFeedPosition:=T_Station.THardware.TAxisToolFeeder.T_LiveValue.lrActualPosition - rActualToolFeederPosition1;
			T_Visu.ptrT_ExchgParam^.T_InfoValueCommon.rActualWireFeedSpeed:=T_Station.THardware.TAxisToolFeeder.T_LiveValue.lrActualVelocity;
		END_IF;
	END_IF;
	T_Visu.ptrT_ExchgParam^.T_InfoValueCommon.rActualGrindAxisPosition:=T_Station.THardware.TAxisGrindFeeder.T_LiveValue.lrActualPosition;
	T_Visu.ptrT_ExchgParam^.T_InfoValueCommon.rActualGrindAxisSpeed:=T_Station.THardware.TAxisGrindFeeder.T_LiveValue.lrActualVelocity;
	T_Visu.ptrT_ExchgParam^.T_StationCommon.rActualGrindFeederPosition:=T_Station.THardware.TAxisGrindFeeder.T_LiveValue.lrActualPosition;
	T_Visu.ptrT_ExchgParam^.T_StationCommon.rActualGrindSpindleSpeed:=T_Station.THardware.TAxisGrindSpindle.T_LiveValue.lrActualVelocity;
	T_Visu.ptrT_ExchgParam^.T_StationCommon.iGrindSpindleLoad:=T_Station.THardware.TAxisGrindSpindle.T_LiveValue.uiActualTorque;
	T_Visu.ptrT_ExchgParam^.T_StationCommon.rGrindSpindleTiltSensor:=T_Station.THardware.TAxisGrindSpindle.T_LiveValue.lrActualPosition;
	T_Visu.ptrT_ExchgParam^.T_StationCommon.xGrindSpindleCW:=NOT(QxGrindingSpindle_CCW);

	IF (T_Visu.ptrT_ExchgParam^.T_TeachIn.iSaveToolFeederPos = 0) THEN
		T_Visu.ptrT_ExchgParam^.T_StationCommon.rOldToolFeederPosition:=0.0;
	END_IF;
	IF (T_Visu.ptrT_ExchgParam^.T_TeachIn.iSaveToolFeederPos = 1) THEN
		T_Visu.ptrT_ExchgParam^.T_StationCommon.rOldToolFeederPosition:=T_NovRam.T_Data.T_ProcessImageData.T_ProcessPara.rStartPosToolFeedAuto;
	END_IF;
	IF (T_Visu.ptrT_ExchgParam^.T_TeachIn.iSaveToolFeederPos = 2) THEN
		T_Visu.ptrT_ExchgParam^.T_StationCommon.rOldToolFeederPosition:=T_NovRam.T_Data.T_ProcessImageData.T_CalibrationPara.rStartPosToolFeedCalib;
	END_IF;
	IF (T_Visu.ptrT_ExchgParam^.T_TeachIn.iSaveToolFeederPos = 3) THEN
		T_Visu.ptrT_ExchgParam^.T_StationCommon.rOldToolFeederPosition:=T_NovRam.T_Data.T_ProcessImageData.T_CalibrationPara.rMeasurePosToolFeedCalib;
	END_IF;
	IF (T_Visu.ptrT_ExchgParam^.T_TeachIn.iSaveToolFeederPos = 4) THEN
		T_Visu.ptrT_ExchgParam^.T_StationCommon.rOldToolFeederPosition:=T_NovRam.T_Data.T_Standard.T_AxisPosition.rLoadPosToolFeedAuto;
	END_IF;
	IF (T_Visu.ptrT_ExchgParam^.T_TeachIn.iSaveGrindFeederPos = 0) THEN
		T_Visu.ptrT_ExchgParam^.T_StationCommon.rOldGrindFeederPosition:=0.0;
	END_IF;
	IF (T_Visu.ptrT_ExchgParam^.T_TeachIn.iSaveGrindFeederPos = 1) THEN
		T_Visu.ptrT_ExchgParam^.T_StationCommon.rOldGrindFeederPosition:=T_NovRam.T_Data.T_ProcessImageData.T_ProcessPara.rToolDiameterProcess;
	END_IF;
	IF (T_Visu.ptrT_ExchgParam^.T_TeachIn.iSaveGrindFeederPos = 2) THEN
		(* Security Position will be calculateted with the settled Tooldiameter plus the Offset *)
		T_Visu.ptrT_ExchgParam^.T_StationCommon.rOldGrindFeederPosition:=	T_NovRam.T_Data.T_ProcessImageData.T_ProcessPara.rToolDiameterProcess +
																		T_NovRam.T_Data.T_ProcessImageData.T_ProcessPara.rSecurityPosGrindFeedProcess;
	END_IF;
	IF (T_Visu.ptrT_ExchgParam^.T_TeachIn.iSaveGrindFeederPos = 3) THEN
		T_Visu.ptrT_ExchgParam^.T_StationCommon.rOldGrindFeederPosition:=T_NovRam.T_Data.T_ProcessImageData.T_PrismPara.rToolDiameterMin;
	END_IF;
	IF (T_Visu.ptrT_ExchgParam^.T_TeachIn.iSaveGrindFeederPos = 4) THEN
		T_Visu.ptrT_ExchgParam^.T_StationCommon.rOldGrindFeederPosition:=T_NovRam.T_Data.T_ProcessImageData.T_PrismPara.rToolDiameterMax + T_NovRam.T_Data.T_Standard.T_TeachINGrindFeeder.rOffsetSWPosEndSwitch;
	END_IF;

(* Monitoring Cylinder value *)
	(* Cyl ToolTension *)
	T_Visu.ptrT_ExchgParam^.T_Cylinder.xToolTension:=T_Station.THardware.TCylToolTension.T_CtrleCyl.T_AnalogCylinder.xActiv;
	IF T_Station.THardware.TCylToolTension.T_CtrleCyl.xStatePosOn THEN T_Visu.ptrT_ExchgParam^.T_Cylinder.bPosToolTension:=T_Visu.ptrT_ExchgParam^.T_Cylinder.bPosToolTension OR 16#1;
		ELSE T_Visu.ptrT_ExchgParam^.T_Cylinder.bPosToolTension:=T_Visu.ptrT_ExchgParam^.T_Cylinder.bPosToolTension AND 16#FE; END_IF
	IF (T_Visu.ptrT_ExchgParam^.T_Cylinder.iSelectToolTensionForce < 2) THEN
		T_Visu.ptrT_ExchgParam^.T_Cylinder.rToSetToolTensionForce:=T_NovRam.T_Data.T_ProcessImageData.T_ProcessPara.rToolTensionProcess;
	END_IF;
	IF (T_Visu.ptrT_ExchgParam^.T_Cylinder.iSelectToolTensionForce > 1) THEN
		T_Visu.ptrT_ExchgParam^.T_Cylinder.rToSetToolTensionForce:=T_NovRam.T_Data.T_Standard.T_Cyl_ToolTension.rForce;
	END_IF;
	(*22.12.2009: KFS	{	 *)
	IF xMicroRodActive THEN
		(* Cyl ToolLeft *)
		T_Visu.ptrT_ExchgParam^.T_Cylinder.xCylToolLeft:=T_Station.THardware.TCylToolLeftActive.T_CtrleCyl.T_Standard.xActivOn;
		IF T_Station.THardware.TCylToolLeftActive.T_CtrleCyl.xStatePosOn THEN T_Visu.ptrT_ExchgParam^.T_Cylinder.bPosCylToolLeft:=T_Visu.ptrT_ExchgParam^.T_Cylinder.bPosCylToolLeft OR 16#1;
			ELSE T_Visu.ptrT_ExchgParam^.T_Cylinder.bPosCylToolLeft:=T_Visu.ptrT_ExchgParam^.T_Cylinder.bPosCylToolLeft AND 16#FE; END_IF
		IF T_Station.THardware.TCylToolLeftActive.T_CtrleCyl.xStatePosOff THEN T_Visu.ptrT_ExchgParam^.T_Cylinder.bPosCylToolLeft:=T_Visu.ptrT_ExchgParam^.T_Cylinder.bPosCylToolLeft OR 16#2;
			ELSE T_Visu.ptrT_ExchgParam^.T_Cylinder.bPosCylToolLeft:=T_Visu.ptrT_ExchgParam^.T_Cylinder.bPosCylToolLeft AND 16#FD; END_IF
		(* Cyl ToolRight *)
		T_Visu.ptrT_ExchgParam^.T_Cylinder.xCylToolRight:=T_Station.THardware.TCylToolRightActive.T_CtrleCyl.T_Standard.xActivOn;
		IF T_Station.THardware.TCylToolRightActive.T_CtrleCyl.xStatePosOn THEN T_Visu.ptrT_ExchgParam^.T_Cylinder.bPosCylToolRight:=T_Visu.ptrT_ExchgParam^.T_Cylinder.bPosCylToolRight OR 16#1;
			ELSE T_Visu.ptrT_ExchgParam^.T_Cylinder.bPosCylToolRight:=T_Visu.ptrT_ExchgParam^.T_Cylinder.bPosCylToolRight AND 16#FE; END_IF
		IF T_Station.THardware.TCylToolRightActive.T_CtrleCyl.xStatePosOff THEN T_Visu.ptrT_ExchgParam^.T_Cylinder.bPosCylToolRight:=T_Visu.ptrT_ExchgParam^.T_Cylinder.bPosCylToolRight OR 16#2;
			ELSE T_Visu.ptrT_ExchgParam^.T_Cylinder.bPosCylToolRight:=T_Visu.ptrT_ExchgParam^.T_Cylinder.bPosCylToolRight AND 16#FD; END_IF
		(* Cyl ToolCenter *)
		T_Visu.ptrT_ExchgParam^.T_Cylinder.xCylToolCenter:=T_Station.THardware.TCylToolCenterActive.T_CtrleCyl.T_Standard.xActivOn;
		IF T_Station.THardware.TCylToolCenterActive.T_CtrleCyl.xStatePosOn THEN T_Visu.ptrT_ExchgParam^.T_Cylinder.bPosCylToolCenter:=T_Visu.ptrT_ExchgParam^.T_Cylinder.bPosCylToolCenter OR 16#1;
			ELSE T_Visu.ptrT_ExchgParam^.T_Cylinder.bPosCylToolCenter:=T_Visu.ptrT_ExchgParam^.T_Cylinder.bPosCylToolCenter AND 16#FE; END_IF
		IF T_Station.THardware.TCylToolCenterActive.T_CtrleCyl.xStatePosOff THEN T_Visu.ptrT_ExchgParam^.T_Cylinder.bPosCylToolCenter:=T_Visu.ptrT_ExchgParam^.T_Cylinder.bPosCylToolCenter OR 16#2;
			ELSE T_Visu.ptrT_ExchgParam^.T_Cylinder.bPosCylToolCenter:=T_Visu.ptrT_ExchgParam^.T_Cylinder.bPosCylToolCenter AND 16#FD; END_IF
		(* Cyl ToolPrismaLeft *)
		T_Visu.ptrT_ExchgParam^.T_Cylinder.xCylToolPrismaLeft:=T_Station.THardware.TCylToolPrismaLeftActive.T_CtrleCyl.T_Standard.xActivOn;
		IF T_Station.THardware.TCylToolPrismaLeftActive.T_CtrleCyl.xStatePosOn THEN T_Visu.ptrT_ExchgParam^.T_Cylinder.bPosCylToolPrismaLeft:=T_Visu.ptrT_ExchgParam^.T_Cylinder.bPosCylToolPrismaLeft OR 16#1;
			ELSE T_Visu.ptrT_ExchgParam^.T_Cylinder.bPosCylToolPrismaLeft:=T_Visu.ptrT_ExchgParam^.T_Cylinder.bPosCylToolPrismaLeft AND 16#FE; END_IF
		IF T_Station.THardware.TCylToolPrismaLeftActive.T_CtrleCyl.xStatePosOff THEN T_Visu.ptrT_ExchgParam^.T_Cylinder.bPosCylToolPrismaLeft:=T_Visu.ptrT_ExchgParam^.T_Cylinder.bPosCylToolPrismaLeft OR 16#2;
			ELSE T_Visu.ptrT_ExchgParam^.T_Cylinder.bPosCylToolPrismaLeft:=T_Visu.ptrT_ExchgParam^.T_Cylinder.bPosCylToolPrismaLeft AND 16#FD; END_IF
		(* Cyl ToolPrismaRight *)
		T_Visu.ptrT_ExchgParam^.T_Cylinder.xCylToolPrismaRight:=T_Station.THardware.TCylToolPrismaRightActive.T_CtrleCyl.T_Standard.xActivOn;
		IF T_Station.THardware.TCylToolPrismaRightActive.T_CtrleCyl.xStatePosOn THEN T_Visu.ptrT_ExchgParam^.T_Cylinder.bPosCylToolPrismalRight:=T_Visu.ptrT_ExchgParam^.T_Cylinder.bPosCylToolPrismalRight OR 16#1;
			ELSE T_Visu.ptrT_ExchgParam^.T_Cylinder.bPosCylToolPrismalRight:=T_Visu.ptrT_ExchgParam^.T_Cylinder.bPosCylToolPrismalRight AND 16#FE; END_IF
		IF T_Station.THardware.TCylToolPrismaRightActive.T_CtrleCyl.xStatePosOff THEN T_Visu.ptrT_ExchgParam^.T_Cylinder.bPosCylToolPrismalRight:=T_Visu.ptrT_ExchgParam^.T_Cylinder.bPosCylToolPrismalRight OR 16#2;
			ELSE T_Visu.ptrT_ExchgParam^.T_Cylinder.bPosCylToolPrismalRight:=T_Visu.ptrT_ExchgParam^.T_Cylinder.bPosCylToolPrismalRight AND 16#FD; END_IF
	END_IF;
	(*22.12.2009: KFS	}	 *)
END_ACTION
ACTION VisuFunction_Axis:
(* Action stop axis *)
	IF xStopAxis THEN
		(* Step stop axis *)
		CASE iStepAction OF
		(* check axis *)
		1:	xMoveAbsPosition:=xMoveRelPosition:=xMoveContinousVel:=FALSE;
			IF NOT T_Station.TControl.xHardwareConfigError THEN
				xStepActionDone:=FALSE;
				IF ptrTeachINAxis^.T_CtrleSingle.xErr THEN
					iStepAction:=99;
					RETURN;
				END_IF;
				iStepAction:=95;
				xTmp:=	ptrTeachINAxis^.T_CtrleSingle.xReady (*AND
						NOT(ptrTeachINAxis^.T_CtrleSingle.xErr)*);
				(* Start/Stop position or speed of teachin page has to be confirmed *)
				IF xTmp THEN
					iStepAction:=10;
				ELSE
					iStepAction:=95;
				END_IF
			ELSE
				iStepAction:=95;
			END_IF;
		(* activ function axis *)
		10:	ptrTeachINAxis^.T_CtrleSingle.iFunction:=5;
			ptrTeachINAxis^.T_CtrleSingle.xExecute:=TRUE;
			(* init. acc/dec/jerk *)
			ptrTeachINAxis^.T_CtrleSingle.lrAcceleration:=TParaAxisTeachIN.rAcceleration;
			ptrTeachINAxis^.T_CtrleSingle.lrDecceleration:=TParaAxisTeachIN.rDeceleration;
			(*
			ptrTeachINAxis^.T_CtrleSingle.lrAcceleration:=ptrTeachINAxis^.T_Config_ObjFileValue.lrAcceleration;
			ptrTeachINAxis^.T_CtrleSingle.lrDecceleration:=ptrTeachINAxis^.T_Config_ObjFileValue.lrDecceleration;
			ptrTeachINAxis^.T_CtrleSingle.lrJerk:=ptrTeachINAxis^.T_Config_ObjFileValue.lrJerk;
			*)
			(* next step *)
			iStepAction:=20;
			xStepActionDone:=FALSE;
		(* waiting stop confirmation *)
		20:	IF NOT(xStepActionDone) THEN
			(* confirm execution *)
				ptrTeachINAxis^.T_CtrleSingle.xExecute:=FALSE;
				xStepActionDone:=TRUE;
			ELSE
				IF ptrTeachINAxis^.T_CtrleSingle.xDone THEN
				(* confirm action next step *)
					iStepAction:=90;
					xStepActionDone:=FALSE;
				ELSE
					IF ptrTeachINAxis^.T_CtrleSingle.xErr THEN
					(* activ action not ready or error *)
						iStepAction:=99;
						xStepActionDone:=FALSE;
					END_IF
				END_IF
			END_IF
		(* waiting time out *)
		89:	IF TimerAction.Q THEN iStepAction:=90; END_IF
			(*T_Visu.ptrT_ExchgParam^.T_TeachIn.iStateAxisMovement:=1;*)
		(* action done *)
		90:	bStateMachine:=1;
			xSetStateMachine:=TRUE;
			T_Visu.ptrT_ExchgParam^.T_StationCommon.wState:=T_Visu.ptrT_ExchgParam^.T_StationCommon.wState AND 16#BF;
			T_Visu.T_CtrleAction.xDone:=TRUE;
			T_Visu.T_CtrleAction.xNotReady:=FALSE;
			T_Visu.T_CtrleAction.xErr:=FALSE;
			T_Visu.T_CtrleAction.udiErrorID:=0;
			xStopAxis:=FALSE;
			(*T_Visu.ptrT_ExchgParam^.T_TeachIn.iStateAxisMovement:=1;*)
		(* axis not ready *)
		95:	T_Visu.ptrT_ExchgParam^.T_StationCommon.wState:=T_Visu.ptrT_ExchgParam^.T_StationCommon.wState AND 16#BF;
			TimerNotReady(IN:=TRUE);
			xStopAxis:=FALSE;
			(*T_Visu.ptrT_ExchgParam^.T_TeachIn.iStateAxisMovement:=1;*)
		(* error *)
		99:	T_Visu.ptrT_ExchgParam^.T_StationCommon.wState:=T_Visu.ptrT_ExchgParam^.T_StationCommon.wState AND 16#BF;
			T_Visu.T_CtrleAction.xDone:=TRUE;
			T_Visu.T_CtrleAction.xNotReady:=FALSE;
			IF (ptrTeachINAxis^.T_Config_Gen.iTyp <> 0) THEN
				diErrorNr:=(ptrTeachINAxis^.T_Config_Gen.iTyp * 1000000) + ptrTeachINAxis^.T_CtrleSingle.udiErrorID;
			ELSE
				diErrorNr:=0;
			END_IF;
			FBErrorMessage(	diErrorNr:=diErrorNr,
							T_ErrorList:=T_ErrorList);
			T_Visu.ptrT_ExchgParam^.T_Visu.T_Message.sDynamicTextEnglish:=FBErrorMessage.sErrorTextEnglish;
			T_Visu.ptrT_ExchgParam^.T_Visu.T_Message.sDynamicTextDeutsch:=FBErrorMessage.sErrorTextDeutsch;
			T_Visu.ptrT_ExchgParam^.T_Visu.T_Message.sDynamicTextFrancais:=FBErrorMessage.sErrorTextFrancais;
			T_Visu.ptrT_ExchgParam^.T_SafetyCtrl.xSetForceError:=TRUE;
			T_Visu.ptrT_ExchgParam^.T_SafetyCtrl.diSetForceErrorNr:=diErrorNr;
			T_Visu.T_CtrleAction.xErr:=FALSE;
			T_Visu.T_CtrleAction.udiErrorID:=0;
			ptrTeachINAxis^.T_CtrleSingle.iFunction:=1;
			ptrTeachINAxis^.T_CtrleSingle.xExecute:=TRUE;
			xStopAxis:=FALSE;
			T_StartUp.T_Ctrle.xSetSecurityStateON:=TRUE;
		END_CASE
	END_IF

(* Action move abs position *)
	IF xMoveAbsPosition OR xMoveRelPosition THEN
		(* Step move abs position *)
		CASE iStepAction OF
		(* check axis *)
		1:	IF NOT T_Station.TControl.xHardwareConfigError THEN
				xStepActionDone:=FALSE;
				iStepAction:=95;
				xTmp:=	ptrTeachINAxis^.T_CtrleSingle.xDone
						AND ptrTeachINAxis^.T_CtrleSingle.xReady
						AND ptrTeachINAxis^.T_CtrleSingle.xNotMoving
						AND ptrTeachINAxis^.T_CtrleSingle.xPower
						AND NOT(ptrTeachINAxis^.T_CtrleSingle.xErr)
						AND NOT(ptrTeachINAxis^.T_CtrleSingle.xExecute)
(*24.09.2010: KFS	{	 *)
						AND( (  T_Visu.T_PlcParam.dwActualPage = 210
							   AND NOT(T_Station.THardware.TCylToolLeftActive.T_CtrleCyl.T_Standard.xActivOn)
							   AND NOT(T_Station.THardware.TCylToolRightActive.T_CtrleCyl.T_Standard.xActivOn)
					     		   AND NOT(T_Station.THardware.TCylToolCenterActive.T_CtrleCyl.T_Standard.xActivOn) )  OR ( T_Visu.T_PlcParam.dwActualPage <> 210))
(*24.09.2010: KFS	}	 *)
						AND ((ptrTeachINAxis^.T_CtrleSingle.xRef AND xMoveAbsPosition AND xMicroRodActive) OR NOT(xMicroRodActive)OR xMoveRelPosition);
				(* Start/Stop position or speed of teachin page has to be confirmed *)
				IF xTmp THEN
					iStepAction:=10;
				ELSE
					IF NOT ptrTeachINAxis^.T_CtrleSingle.xRef AND xMoveAbsPosition THEN
					(* Display message, axis not referenced *)
						tTimeOutAction:=TimerAction.ET+T#2s;
						T_Visu.ptrT_ExchgParam^.T_Visu.T_Message.iState:=18;
						(* Action has been cancelled *)
						iStepAction:=89;
					END_IF
				END_IF
			ELSE
				iStepAction:=95;
			END_IF;
		(* activ function axis *)
		10:	tTimeOutAction:=T#999s;
			bStateMachine:=2;
			xSetStateMachine:=TRUE;
			IF xMoveAbsPosition THEN iStepAction:=20; END_IF
			IF xMoveRelPosition THEN iStepAction:=35; END_IF
			(* init. acc/dec/jerk *)
			ptrTeachINAxis^.T_CtrleSingle.lrAcceleration:=TParaAxisTeachIN.rAcceleration;
			ptrTeachINAxis^.T_CtrleSingle.lrDecceleration:=TParaAxisTeachIN.rDeceleration;
			(*
			ptrTeachINAxis^.T_CtrleSingle.lrAcceleration:=ptrTeachINAxis^.T_Config_ObjFileValue.lrAcceleration;
			ptrTeachINAxis^.T_CtrleSingle.lrDecceleration:=ptrTeachINAxis^.T_Config_ObjFileValue.lrDecceleration;
			ptrTeachINAxis^.T_CtrleSingle.lrJerk:=ptrTeachINAxis^.T_Config_ObjFileValue.lrJerk;
			*)
		(* activ function axis move absolut *)
		20:	ptrTeachINAxis^.T_CtrleSingle.iFunction:=7;
			ptrTeachINAxis^.T_CtrleSingle.xExecute:=TRUE;
			(* next step *)
			iStepAction:=40;
			xStepActionDone:=FALSE;
		(* activ function axis move relativ *)
		35:	ptrTeachINAxis^.T_CtrleSingle.iFunction:=8;
			ptrTeachINAxis^.T_CtrleSingle.xExecute:=TRUE;
			(* next step *)
			iStepAction:=40;
			xStepActionDone:=FALSE;
		(* confirm execution *)
		40:	IF NOT(xStepActionDone) THEN
			(* confirm execution *)
				ptrTeachINAxis^.T_CtrleSingle.xExecute:=FALSE;
				xStepActionDone:=TRUE;
				(* Display message, 'Start moving' *)
				T_Visu.ptrT_ExchgParam^.T_Visu.T_Message.iState:=26;
			ELSE
				IF ptrTeachINAxis^.T_CtrleSingle.xDone THEN
				(* confirm action next step *)
					bStateMachine:=1;
					xSetStateMachine:=TRUE;
					iStepAction:=90;
					xStepActionDone:=FALSE;
				ELSE
					IF ptrTeachINAxis^.T_CtrleSingle.xErr THEN
					(* activ action not ready or error *)
						iStepAction:=99;
						xStepActionDone:=FALSE;
					END_IF
				END_IF
			END_IF
		(* waiting timeout *)
		89: IF TimerAction.Q THEN iStepAction:=90; END_IF
			(*T_Visu.ptrT_ExchgParam^.T_TeachIn.iStateAxisMovement:=1;*)
		(* action done *)
		90:	T_Visu.ptrT_ExchgParam^.T_StationCommon.wState:=T_Visu.ptrT_ExchgParam^.T_StationCommon.wState AND 16#BF;
			T_Visu.T_CtrleAction.xDone:=TRUE;
			T_Visu.T_CtrleAction.xNotReady:=FALSE;
			T_Visu.T_CtrleAction.xErr:=FALSE;
			T_Visu.T_CtrleAction.udiErrorID:=0;
			xMoveAbsPosition:=FALSE;
			xMoveRelPosition:=FALSE;
			(*T_Visu.ptrT_ExchgParam^.T_TeachIn.iStateAxisMovement:=1;*)
		(* axis not ready *)
		95:	T_Visu.ptrT_ExchgParam^.T_StationCommon.wState:=T_Visu.ptrT_ExchgParam^.T_StationCommon.wState AND 16#BF;
			TimerNotReady(IN:=TRUE);
			xMoveAbsPosition:=FALSE;
			xMoveRelPosition:=FALSE;
			(*T_Visu.ptrT_ExchgParam^.T_TeachIn.iStateAxisMovement:=1;*)
		(* error *)
		99:	T_Visu.ptrT_ExchgParam^.T_StationCommon.wState:=T_Visu.ptrT_ExchgParam^.T_StationCommon.wState AND 16#BF;
			T_Visu.T_CtrleAction.xDone:=TRUE;
			T_Visu.T_CtrleAction.xNotReady:=FALSE;
			IF (ptrTeachINAxis^.T_Config_Gen.iTyp <> 0) THEN
				diErrorNr:=(ptrTeachINAxis^.T_Config_Gen.iTyp * 1000000) + ptrTeachINAxis^.T_CtrleSingle.udiErrorID;
			ELSE
				diErrorNr:=0;
			END_IF;
			FBErrorMessage(	diErrorNr:=diErrorNr,
							T_ErrorList:=T_ErrorList);
			T_Visu.ptrT_ExchgParam^.T_Visu.T_Message.sDynamicTextEnglish:=FBErrorMessage.sErrorTextEnglish;
			T_Visu.ptrT_ExchgParam^.T_Visu.T_Message.sDynamicTextDeutsch:=FBErrorMessage.sErrorTextDeutsch;
			T_Visu.ptrT_ExchgParam^.T_Visu.T_Message.sDynamicTextFrancais:=FBErrorMessage.sErrorTextFrancais;
			T_Visu.ptrT_ExchgParam^.T_SafetyCtrl.xSetForceError:=TRUE;
			T_Visu.ptrT_ExchgParam^.T_SafetyCtrl.diSetForceErrorNr:=diErrorNr;
			T_Visu.T_CtrleAction.xErr:=FALSE;
			T_Visu.T_CtrleAction.udiErrorID:=0;
			ptrTeachINAxis^.T_CtrleSingle.iFunction:=1;
			ptrTeachINAxis^.T_CtrleSingle.xExecute:=TRUE;
			xMoveAbsPosition:=FALSE;
			xMoveRelPosition:=FALSE;
			T_StartUp.T_Ctrle.xSetSecurityStateON:=TRUE;
			(*T_Visu.ptrT_ExchgParam^.T_TeachIn.iStateAxisMovement:=1;*)
		END_CASE
	END_IF

(* Action move velocity *)
	IF xMoveContinousVel THEN
		(* Step move continuous velocity *)
		CASE iStepAction OF
		(* check axis *)
		1:	IF NOT T_Station.TControl.xHardwareConfigError THEN
				xStepActionDone:=FALSE;
				iStepAction:=95;
				xTmp:=	ptrTeachINAxis^.T_CtrleSingle.xDone
						AND ptrTeachINAxis^.T_CtrleSingle.xReady
						AND ptrTeachINAxis^.T_CtrleSingle.xNotMoving
						AND ptrTeachINAxis^.T_CtrleSingle.xPower
						AND NOT(ptrTeachINAxis^.T_CtrleSingle.xErr)
						AND NOT(ptrTeachINAxis^.T_CtrleSingle.xExecute)
(*24.09.2010: KFS	{	 *)
						AND( (  T_Visu.T_PlcParam.dwActualPage = 210
							   AND NOT(T_Station.THardware.TCylToolLeftActive.T_CtrleCyl.T_Standard.xActivOn)
							   AND NOT(T_Station.THardware.TCylToolRightActive.T_CtrleCyl.T_Standard.xActivOn)
					     		   AND NOT(T_Station.THardware.TCylToolCenterActive.T_CtrleCyl.T_Standard.xActivOn) )  OR ( T_Visu.T_PlcParam.dwActualPage <> 210))
(*24.09.2010: KFS	}	 *)
						AND (ptrTeachINAxis^.T_CtrleSingle.lrVelocity <> 0);
				(* Start/Stop position or speed of teachin page has to be confirmed *)
				IF xTmp THEN
					iStepAction:=10;
				END_IF
			ELSE
				iStepAction:=95;
			END_IF;
		(* activ function axis *)
		10:	IF (iSelectedAxis <> 6) THEN	(* IGS *)
				bStateMachine:=2;
			END_IF
			xSetStateMachine:=TRUE;
			ptrTeachINAxis^.T_CtrleSingle.iFunction:=6;
			ptrTeachINAxis^.T_CtrleSingle.xExecute:=TRUE;
			(* init. acc/dec/jerk *)
			ptrTeachINAxis^.T_CtrleSingle.lrAcceleration:=TParaAxisTeachIN.rAcceleration;
			ptrTeachINAxis^.T_CtrleSingle.lrDecceleration:=TParaAxisTeachIN.rDeceleration;
			(*
			ptrTeachINAxis^.T_CtrleSingle.lrAcceleration:=ptrTeachINAxis^.T_Config_ObjFileValue.lrAcceleration;
			ptrTeachINAxis^.T_CtrleSingle.lrDecceleration:=ptrTeachINAxis^.T_Config_ObjFileValue.lrDecceleration;
			ptrTeachINAxis^.T_CtrleSingle.lrJerk:=ptrTeachINAxis^.T_Config_ObjFileValue.lrJerk;
			*)
			(* next step *)
			iStepAction:=20;
			xStepActionDone:=FALSE;
		(* confirm execution *)
		20:	IF NOT(xStepActionDone) THEN
			(* confirm execution *)
				ptrTeachINAxis^.T_CtrleSingle.xExecute:=FALSE;
				xStepActionDone:=TRUE;
			ELSE
				IF ptrTeachINAxis^.T_CtrleSingle.xDone THEN
				(* confirm action next step *)
					iStepAction:=90;
					xStepActionDone:=FALSE;
				ELSE
					IF ptrTeachINAxis^.T_CtrleSingle.xErr THEN
					(* activ action not ready or error *)
						iStepAction:=99;
						xStepActionDone:=FALSE;
					END_IF
				END_IF
			END_IF
		(* action done *)
		90:	T_Visu.ptrT_ExchgParam^.T_StationCommon.wState:=T_Visu.ptrT_ExchgParam^.T_StationCommon.wState AND 16#BF;
			T_Visu.T_CtrleAction.xDone:=TRUE;
			T_Visu.T_CtrleAction.xNotReady:=FALSE;
			T_Visu.T_CtrleAction.xErr:=FALSE;
			T_Visu.T_CtrleAction.udiErrorID:=0;
			xMoveContinousVel:=FALSE;
		(* axis not ready *)
		95:	T_Visu.ptrT_ExchgParam^.T_StationCommon.wState:=T_Visu.ptrT_ExchgParam^.T_StationCommon.wState AND 16#BF;
			TimerNotReady(IN:=TRUE);
			xMoveContinousVel:=FALSE;
		(* error *)
		99:	T_Visu.ptrT_ExchgParam^.T_StationCommon.wState:=T_Visu.ptrT_ExchgParam^.T_StationCommon.wState AND 16#BF;
			T_Visu.T_CtrleAction.xDone:=TRUE;
			T_Visu.T_CtrleAction.xNotReady:=FALSE;
			IF (ptrTeachINAxis^.T_Config_Gen.iTyp <> 0) THEN
				diErrorNr:=(ptrTeachINAxis^.T_Config_Gen.iTyp * 1000000) + ptrTeachINAxis^.T_CtrleSingle.udiErrorID;
			ELSE
				diErrorNr:=0;
			END_IF;
			FBErrorMessage(	diErrorNr:=diErrorNr,
							T_ErrorList:=T_ErrorList);
			T_Visu.ptrT_ExchgParam^.T_Visu.T_Message.sDynamicTextEnglish:=FBErrorMessage.sErrorTextEnglish;
			T_Visu.ptrT_ExchgParam^.T_Visu.T_Message.sDynamicTextDeutsch:=FBErrorMessage.sErrorTextDeutsch;
			T_Visu.ptrT_ExchgParam^.T_Visu.T_Message.sDynamicTextFrancais:=FBErrorMessage.sErrorTextFrancais;
			T_Visu.ptrT_ExchgParam^.T_SafetyCtrl.xSetForceError:=TRUE;
			T_Visu.ptrT_ExchgParam^.T_SafetyCtrl.diSetForceErrorNr:=diErrorNr;
			T_Visu.T_CtrleAction.xErr:=FALSE;
			T_Visu.T_CtrleAction.udiErrorID:=0;
			ptrTeachINAxis^.T_CtrleSingle.iFunction:=1;
			ptrTeachINAxis^.T_CtrleSingle.xExecute:=TRUE;
			xMoveContinousVel:=FALSE;
		END_CASE
	END_IF

(* Action Toggle Axis Power *)
	IF xToggleAxisPower OR xResetAxis THEN
		(* Step toggle Axis power *)
		CASE iStepAction OF
		(* check axis *)
		1:	IF NOT T_Station.TControl.xHardwareConfigError THEN
				xStepActionDone:=FALSE;
				iStepAction:=95;
				IF xToggleAxisPower THEN
					xTmp:=	ptrTeachINAxis^.T_CtrleSingle.xDone
							AND ptrTeachINAxis^.T_CtrleSingle.xNotMoving
							AND NOT(ptrTeachINAxis^.T_CtrleSingle.xErr)
							AND NOT(ptrTeachINAxis^.T_CtrleSingle.xExecute);
				END_IF;
				IF xResetAxis THEN
					xTmp:=	(ptrTeachINAxis^.T_CtrleSingle.xDone OR ptrTeachINAxis^.T_CtrleSingle.xErr)
							AND ptrTeachINAxis^.T_CtrleSingle.xNotMoving
							AND NOT(ptrTeachINAxis^.T_CtrleSingle.xExecute);
				END_IF;
				(* Start/Stop position or speed of teachin page has to be confirmed *)
				IF xTmp THEN
					iStepAction:=10;
				END_IF
			ELSE
				iStepAction:=95;
			END_IF;
		(* activ function axis *)
		10:	bStateMachine:=2;
			xSetStateMachine:=TRUE;
			IF xToggleAxisPower THEN
				IF ptrTeachINAxis^.T_CtrleSingle.xPower THEN
					ptrTeachINAxis^.T_CtrleSingle.iFunction:=4;
				END_IF;
				IF NOT(ptrTeachINAxis^.T_CtrleSingle.xPower) THEN
					ptrTeachINAxis^.T_CtrleSingle.iFunction:=3;
				END_IF;
			END_IF;
			IF xResetAxis THEN
				ptrTeachINAxis^.T_CtrleSingle.iFunction:=1;
			END_IF;
			ptrTeachINAxis^.T_CtrleSingle.xExecute:=TRUE;
			(* next step *)
			iStepAction:=20;
			xStepActionDone:=FALSE;
		(* confirm execution *)
		20:	IF NOT(xStepActionDone) THEN
			(* confirm execution *)
				ptrTeachINAxis^.T_CtrleSingle.xExecute:=FALSE;
				xStepActionDone:=TRUE;
			ELSE
				IF ptrTeachINAxis^.T_CtrleSingle.xDone THEN
				(* confirm action next step *)
					bStateMachine:=1;
					xSetStateMachine:=TRUE;
					iStepAction:=90;
					xStepActionDone:=FALSE;
				ELSE
					IF ptrTeachINAxis^.T_CtrleSingle.xErr THEN
					(* activ action not ready or error *)
						iStepAction:=99;
						xStepActionDone:=FALSE;
					END_IF
				END_IF
			END_IF
		(* action done *)
		90:	T_Visu.ptrT_ExchgParam^.T_StationCommon.wState:=T_Visu.ptrT_ExchgParam^.T_StationCommon.wState AND 16#BF;
			T_Visu.T_CtrleAction.xDone:=TRUE;
			T_Visu.T_CtrleAction.xNotReady:=FALSE;
			T_Visu.T_CtrleAction.xErr:=FALSE;
			T_Visu.T_CtrleAction.udiErrorID:=0;
			xToggleAxisPower:=xResetAxis:=FALSE;
		(* axis not ready *)
		95:	T_Visu.ptrT_ExchgParam^.T_StationCommon.wState:=T_Visu.ptrT_ExchgParam^.T_StationCommon.wState AND 16#BF;
			TimerNotReady(IN:=TRUE);
			xToggleAxisPower:=xResetAxis:=FALSE;
		(* error *)
		99:	T_Visu.ptrT_ExchgParam^.T_StationCommon.wState:=T_Visu.ptrT_ExchgParam^.T_StationCommon.wState AND 16#BF;
			T_Visu.T_CtrleAction.xDone:=TRUE;
			T_Visu.T_CtrleAction.xNotReady:=FALSE;
			IF (ptrTeachINAxis^.T_Config_Gen.iTyp <> 0) THEN
				diErrorNr:=(ptrTeachINAxis^.T_Config_Gen.iTyp * 1000000) + ptrTeachINAxis^.T_CtrleSingle.udiErrorID;
			ELSE
				diErrorNr:=0;
			END_IF;
			FBErrorMessage(	diErrorNr:=diErrorNr,
							T_ErrorList:=T_ErrorList);
			T_Visu.ptrT_ExchgParam^.T_Visu.T_Message.sDynamicTextEnglish:=FBErrorMessage.sErrorTextEnglish;
			T_Visu.ptrT_ExchgParam^.T_Visu.T_Message.sDynamicTextDeutsch:=FBErrorMessage.sErrorTextDeutsch;
			T_Visu.ptrT_ExchgParam^.T_Visu.T_Message.sDynamicTextFrancais:=FBErrorMessage.sErrorTextFrancais;
			T_Visu.ptrT_ExchgParam^.T_SafetyCtrl.xSetForceError:=TRUE;
			T_Visu.ptrT_ExchgParam^.T_SafetyCtrl.diSetForceErrorNr:=diErrorNr;
			T_Visu.T_CtrleAction.xErr:=FALSE;
			T_Visu.T_CtrleAction.udiErrorID:=0;
			ptrTeachINAxis^.T_CtrleSingle.iFunction:=1;
			ptrTeachINAxis^.T_CtrleSingle.xExecute:=TRUE;
			xToggleAxisPower:=xResetAxis:=FALSE;
		END_CASE
	END_IF

(* Reference axis *)
	IF xReferenceAxis THEN
		(* Step reference Axis *)
		CASE iStepAction OF
		(* check axis *)
		1:	IF NOT T_Station.TControl.xHardwareConfigError THEN
				xStepActionDone:=FALSE;
				iStepAction:=95;
				xTmp:=	T_Station.THardware.TAxisToolFeeder.T_CtrleSingle.xDone
						AND T_Station.THardware.TAxisToolFeeder.T_CtrleSingle.xPower
						AND T_Station.THardware.TAxisToolFeeder.T_CtrleSingle.xNotMoving
						AND NOT(T_Station.THardware.TAxisToolFeeder.T_CtrleSingle.xErr)
						AND NOT(T_Station.THardware.TAxisToolFeeder.T_CtrleSingle.xExecute);
				(* Start/Stop position or speed of teachin page has to be confirmed *)
				IF xTmp THEN
					iStepAction:=10;
				END_IF
			ELSE
				iStepAction:=95;
			END_IF;
		(* activ function axis *)
		10:	bStateMachine:=2;
			xSetStateMachine:=TRUE;
			T_Station.THardware.TAxisToolFeeder.T_CtrleSingle.lrHomingMethode:=5;
			T_Station.THardware.TAxisToolFeeder.T_CtrleSingle.lrHomeOffset:=0.0;
			T_Station.THardware.TAxisToolFeeder.T_CtrleSingle.lrHomeSpeedSwitch:=T_NovRAM.T_Data.T_Standard.T_TeachINToolFeeder.rRefSpeed;
			T_Station.THardware.TAxisToolFeeder.T_CtrleSingle.lrHomeSpeedZero:=T_NovRAM.T_Data.T_Standard.T_TeachINToolFeeder.rRefSpeed / 10.0;
			T_Station.THardware.TAxisToolFeeder.T_CtrleSingle.lrHomeAcceleration:=T_NovRAM.T_Data.T_Standard.T_TeachINToolFeeder.rAcceleration;
			T_Station.THardware.TAxisToolFeeder.T_CtrleSingle.iFunction:=9;	(* Reference Axis *)
			T_Station.THardware.TAxisToolFeeder.T_CtrleSingle.xExecute:=TRUE;
			(* next step *)
			iStepAction:=20;
			xStepActionDone:=FALSE;
		(* confirm execution *)
		20:	IF NOT(xStepActionDone) THEN
			(* confirm execution *)
				T_Station.THardware.TAxisToolFeeder.T_CtrleSingle.xExecute:=FALSE;
				xStepActionDone:=TRUE;
			ELSE
				IF T_Station.THardware.TAxisToolFeeder.T_CtrleSingle.xDone THEN
				(* confirm action next step *)
					bStateMachine:=1;
					xSetStateMachine:=TRUE;
					iStepAction:=90;
					xStepActionDone:=FALSE;
				ELSE
					IF T_Station.THardware.TAxisToolFeeder.T_CtrleSingle.xErr THEN
					(* activ action not ready or error *)
						iStepAction:=99;
						xStepActionDone:=FALSE;
					END_IF
				END_IF
			END_IF
		(* action done *)
		90:	T_Visu.ptrT_ExchgParam^.T_StationCommon.wState:=T_Visu.ptrT_ExchgParam^.T_StationCommon.wState AND 16#BF;
			T_Visu.T_CtrleAction.xDone:=TRUE;
			T_Visu.T_CtrleAction.xNotReady:=FALSE;
			T_Visu.T_CtrleAction.xErr:=FALSE;
			T_Visu.T_CtrleAction.udiErrorID:=0;
			xReferenceAxis:=FALSE;
		(* axis not ready *)
		95:	T_Visu.ptrT_ExchgParam^.T_StationCommon.wState:=T_Visu.ptrT_ExchgParam^.T_StationCommon.wState AND 16#BF;
			TimerNotReady(IN:=TRUE);
			xReferenceAxis:=FALSE;
		(* error *)
		99:	T_Visu.ptrT_ExchgParam^.T_StationCommon.wState:=T_Visu.ptrT_ExchgParam^.T_StationCommon.wState AND 16#BF;
			T_Visu.T_CtrleAction.xDone:=TRUE;
			T_Visu.T_CtrleAction.xNotReady:=FALSE;
			IF (T_Station.THardware.TAxisToolFeeder.T_Config_Gen.iTyp <> 0) THEN
				diErrorNr:=(T_Station.THardware.TAxisToolFeeder.T_Config_Gen.iTyp * 1000000) + T_Station.THardware.TAxisToolFeeder.T_CtrleSingle.udiErrorID;
			ELSE
				diErrorNr:=0;
			END_IF;
			FBErrorMessage(	diErrorNr:=diErrorNr,
							T_ErrorList:=T_ErrorList);
			T_Visu.ptrT_ExchgParam^.T_Visu.T_Message.sDynamicTextEnglish:=FBErrorMessage.sErrorTextEnglish;
			T_Visu.ptrT_ExchgParam^.T_Visu.T_Message.sDynamicTextDeutsch:=FBErrorMessage.sErrorTextDeutsch;
			T_Visu.ptrT_ExchgParam^.T_Visu.T_Message.sDynamicTextFrancais:=FBErrorMessage.sErrorTextFrancais;
			T_Visu.ptrT_ExchgParam^.T_SafetyCtrl.xSetForceError:=TRUE;
			T_Visu.ptrT_ExchgParam^.T_SafetyCtrl.diSetForceErrorNr:=diErrorNr;
			T_Visu.T_CtrleAction.xErr:=FALSE;
			T_Visu.T_CtrleAction.udiErrorID:=0;
			T_Station.THardware.TAxisToolFeeder.T_CtrleSingle.iFunction:=1;
			T_Station.THardware.TAxisToolFeeder.T_CtrleSingle.xExecute:=TRUE;
			xReferenceAxis:=FALSE;
		END_CASE
	END_IF
END_ACTION
ACTION VisuFunction_AxisTeach:
(* Teach axis Position *)
	IF xTeachPosition THEN
		CASE iStepAction OF
		(* check axis *)
		1:	IF NOT T_Station.TControl.xHardwareConfigError THEN
				xStepActionDone:=FALSE;
				iStepAction:=10;
			ELSE
				iStepAction:=95;
			END_IF;
		(* Check teachin position *)
		10:	IF (iSelectedAxis = 4) THEN
				IF (T_Visu.ptrT_ExchgParam^.T_TeachIn.iSaveToolFeederPos = 0) THEN
				(* Display message 'Move position can not be teached' *)
					tTimeOutAction:=TimerAction.ET+T#2s;
					T_Visu.ptrT_ExchgParam^.T_Visu.T_Message.iState:=31;
					(* Action has been cancelled *)
					iStepAction:=89;
				ELSE
					iStepAction:=20;
				END_IF
			END_IF;
			IF (iSelectedAxis = 5) THEN
				IF (T_Visu.ptrT_ExchgParam^.T_TeachIn.iSaveGrindFeederPos = 0) THEN
				(* Display message 'Move position can not be teached' *)
					tTimeOutAction:=TimerAction.ET+T#2s;
					T_Visu.ptrT_ExchgParam^.T_Visu.T_Message.iState:=31;
					(* Action has been cancelled *)
					iStepAction:=89;
				(* Software limit switch pos and neg not possible that we can teach this position *)
				ELSIF (T_Visu.ptrT_ExchgParam^.T_TeachIn.iSaveGrindFeederPos = 3) OR (T_Visu.ptrT_ExchgParam^.T_TeachIn.iSaveGrindFeederPos = 4) THEN
				(* Display message 'Selected position can not be teached' *)
					tTimeOutAction:=TimerAction.ET+T#2s;
					T_ExchgParam.T_Visu.T_Message.iState:=30;
					(* Action has been cancelled *)
					iStepAction:=89;
				ELSE
					iStepAction:=20;
				END_IF
			END_IF;
		(* Check if the Axis is referenced *)
		20:	IF (iSelectedAxis = 4) THEN
				xTmp:=	T_Station.TControl.xReferenced;
				IF NOT(xTmp) THEN
					(* Display message 'Axis not referenced' *)
					tTimeOutAction:=TimerAction.ET+T#2s;
					T_Visu.ptrT_ExchgParam^.T_Visu.T_Message.iState:=18;
					(* Action has been cancelled *)
					iStepAction:=89;
				ELSE
					iStepAction:=30;
				END_IF;
			ELSE
				iStepAction:=30;
			END_IF;
		(* Display message to ask for confirmation *)
		30:	T_Visu.ptrT_ExchgParam^.T_Visu.T_Message.iState:=108;
			iStepAction:=40;
		(* waiting for key <Enter> or <Esc> *)
		40:	IF RisingEdgeKeyPanel_Enter.Q THEN iStepAction:=50;
			ELSE IF RisingEdgeKeyPanel_Esc.Q THEN iStepAction:=90; END_IF END_IF
			(* An other message has been displayed, stop teach action *)
			IF T_Visu.ptrT_ExchgParam^.T_Visu.T_Message.iState<>108 THEN iStepAction:=90; END_IF
		50:	IF (iSelectedAxis = 4) AND (T_Visu.ptrT_ExchgParam^.T_TeachIn.iSaveToolFeederPos = 1) THEN
				T_Visu.ptrT_ExchgParam^.T_StationCommon.T_ProcessPara.rStartPosToolFeedAuto:=
					LREAL_TO_REAL(ptrTeachINAxis^.T_LiveValue.lrActualPosition);
			ELSIF (iSelectedAxis = 4) AND (T_Visu.ptrT_ExchgParam^.T_TeachIn.iSaveToolFeederPos = 2) THEN
				T_Visu.ptrT_ExchgParam^.T_StationCommon.T_CalibrationPara.rStartPosToolFeedCalib:=
					LREAL_TO_REAL(ptrTeachINAxis^.T_LiveValue.lrActualPosition);
			ELSIF (iSelectedAxis = 4) AND (T_Visu.ptrT_ExchgParam^.T_TeachIn.iSaveToolFeederPos = 3) THEN
				T_Visu.ptrT_ExchgParam^.T_StationCommon.T_CalibrationPara.rMeasurePosToolFeedCalib:=
					LREAL_TO_REAL(ptrTeachINAxis^.T_LiveValue.lrActualPosition);
			ELSIF (iSelectedAxis = 4) AND (T_Visu.ptrT_ExchgParam^.T_TeachIn.iSaveToolFeederPos = 4) THEN
				T_Visu.ptrT_ExchgParam^.T_TeachIn.TParam_AxisPosition.rLoadPosToolFeedAuto:=
					LREAL_TO_REAL(ptrTeachINAxis^.T_LiveValue.lrActualPosition);
			END_IF;
			iStepAction:=60;
			IF (iSelectedAxis = 5) AND (T_Visu.ptrT_ExchgParam^.T_TeachIn.iSaveGrindFeederPos = 1) THEN
				(* The StartPosition will be set as absolut position for the GrindFeeder Axis *)
				T_Station.THardware.TAxisGrindFeeder.T_CtrleSingle.rSetPosition:=
					T_NovRam.T_Data.T_ProcessImageData.T_ProcessPara.rToolDiameterProcess;
				iStepAction:=80;
			END_IF;
			IF (iSelectedAxis = 5) AND (T_Visu.ptrT_ExchgParam^.T_TeachIn.iSaveGrindFeederPos = 2) THEN
				(* The Security Position will be set as absolut position for the GrindFeeder Axis *)
				T_Station.THardware.TAxisGrindFeeder.T_CtrleSingle.rSetPosition:=
										T_NovRam.T_Data.T_ProcessImageData.T_ProcessPara.rToolDiameterProcess +
										T_NovRam.T_Data.T_ProcessImageData.T_ProcessPara.rSecurityPosGrindFeedProcess;
				iStepAction:=80;
			END_IF;
		60:	xAction_SaveNovRAMWithoutConfirm:=TRUE;
			iStepActionNovRam:=1;
			(* next step *)
			iStepAction:=70;
		70:	IF NOT(xAction_SaveNovRAMWithoutConfirm) THEN
				iStepAction:=90;
			END_IF;
		(* activ function axis *)
		80:	T_Station.THardware.TAxisGrindFeeder.T_CtrleSingle.iFunction:=11;
			T_Station.THardware.TAxisGrindFeeder.T_CtrleSingle.xExecute:=TRUE;
			(* next step *)
			iStepAction:=81;
			xStepActionDone:=FALSE;
		(* confirm execution *)
		81:	IF NOT(xStepActionDone) THEN
			(* confirm execution *)
				T_Station.THardware.TAxisGrindFeeder.T_CtrleSingle.xExecute:=FALSE;
				xStepActionDone:=TRUE;
			ELSE
				IF T_Station.THardware.TAxisGrindFeeder.T_CtrleSingle.xDone THEN
				(* confirm action next step *)
					iStepAction:=90;
					xStepActionDone:=FALSE;
				ELSE
					IF T_Station.THardware.TAxisGrindFeeder.T_CtrleSingle.xErr THEN
					(* activ action not ready or error *)
						iStepAction:=98;
						xStepActionDone:=FALSE;
					END_IF
				END_IF
			END_IF
		(* waiting timeout *)
		89: IF TimerAction.Q THEN iStepAction:=90; END_IF
		(* axis not ready *)
		95:	TimerNotReady(IN:=TRUE);
			xTeachPosition:=FALSE;
		(* slow/fast configuration done *)
		90:	T_Visu.T_CtrleAction.xDone:=TRUE;
			T_Visu.T_CtrleAction.xNotReady:=FALSE;
			T_Visu.T_CtrleAction.xErr:=FALSE;
			T_Visu.T_CtrleAction.udiErrorID:=0;
			xTeachPosition:=FALSE;
		(* axis error *)
		98:	T_Visu.ptrT_ExchgParam^.T_StationCommon.wState:=T_Visu.ptrT_ExchgParam^.T_StationCommon.wState AND 16#BF;
			T_Visu.T_CtrleAction.xDone:=TRUE;
			T_Visu.T_CtrleAction.xNotReady:=FALSE;
			IF (T_Station.THardware.TAxisGrindFeeder.T_Config_Gen.iTyp <> 0) THEN
				diErrorNr:=(T_Station.THardware.TAxisGrindFeeder.T_Config_Gen.iTyp * 1000000) + T_Station.THardware.TAxisGrindFeeder.T_CtrleSingle.udiErrorID;
			ELSE
				diErrorNr:=0;
			END_IF;
			FBErrorMessage(	diErrorNr:=diErrorNr,
							T_ErrorList:=T_ErrorList);
			T_Visu.ptrT_ExchgParam^.T_Visu.T_Message.sDynamicTextEnglish:=FBErrorMessage.sErrorTextEnglish;
			T_Visu.ptrT_ExchgParam^.T_Visu.T_Message.sDynamicTextDeutsch:=FBErrorMessage.sErrorTextDeutsch;
			T_Visu.ptrT_ExchgParam^.T_Visu.T_Message.sDynamicTextFrancais:=FBErrorMessage.sErrorTextFrancais;
			T_Visu.ptrT_ExchgParam^.T_SafetyCtrl.xSetForceError:=TRUE;
			T_Visu.ptrT_ExchgParam^.T_SafetyCtrl.diSetForceErrorNr:=diErrorNr;
			T_Visu.T_CtrleAction.xErr:=FALSE;
			T_Visu.T_CtrleAction.udiErrorID:=0;
			T_Station.THardware.TAxisGrindFeeder.T_CtrleSingle.iFunction:=1;
			T_Station.THardware.TAxisGrindFeeder.T_CtrleSingle.xExecute:=TRUE;
			xTeachPosition:=FALSE;
		99:	T_Visu.T_CtrleAction.xDone:=FALSE;
			T_Visu.T_CtrleAction.xNotReady:=FALSE;
			T_Visu.T_CtrleAction.xErr:=TRUE;
			T_Visu.T_CtrleAction.udiErrorID:=16#F0000 + T_Visu.T_CtrleAction.iFunction;
			xTeachPosition:=FALSE;
		END_CASE
	END_IF

(* Calculate the position between the RefIndex and the RefSensor *)
	IF xCalcAngleRefIndex THEN
		(* Step calc the position between the RefIndex and the RefSensor *)
		CASE iStepAction OF
		(* check axis *)
		1:	IF NOT T_Station.TControl.xHardwareConfigError THEN
				xStepActionDone:=FALSE;
				iStepAction:=10;
			ELSE
				iStepAction:=95;
			END_IF;
		(* check axis state *)
		10:	xStepActionDone:=FALSE;
			xTmp:=	T_Station.THardware.TAxisToolFeeder.T_CtrleSingle.xDone
					AND T_Station.THardware.TAxisToolFeeder.T_CtrleSingle.xReady
					AND T_Station.THardware.TAxisToolFeeder.T_CtrleSingle.xNotMoving
					AND NOT(T_Station.THardware.TAxisToolFeeder.T_CtrleSingle.xErr)
					AND NOT(T_Station.THardware.TAxisToolFeeder.T_CtrleSingle.xExecute);
			IF xTmp THEN
				iStepAction:=20;
			ELSE
				iStepAction:=95;
			END_IF
		(* activ function axis *)
		20:	bStateMachine:=2;
			xSetStateMachine:=TRUE;
			T_Station.THardware.TAxisToolFeeder.T_CtrleSingle.lrHomingMethode:=5;
			T_Station.THardware.TAxisToolFeeder.T_CtrleSingle.lrHomeOffset:=0.0;
			T_Station.THardware.TAxisToolFeeder.T_CtrleSingle.lrHomeSpeedSwitch:=T_NovRAM.T_Data.T_Standard.T_TeachINToolFeeder.rRefSpeed;
			T_Station.THardware.TAxisToolFeeder.T_CtrleSingle.lrHomeSpeedZero:=T_NovRAM.T_Data.T_Standard.T_TeachINToolFeeder.rRefSpeed / 10.0;
			T_Station.THardware.TAxisToolFeeder.T_CtrleSingle.lrHomeAcceleration:=T_NovRAM.T_Data.T_Standard.T_TeachINToolFeeder.rAcceleration;
			T_Station.THardware.TAxisToolFeeder.T_CtrleSingle.lrDecceleration:=T_NovRAM.T_Data.T_Standard.T_TeachINToolFeeder.rDeceleration;
			T_Station.THardware.TAxisToolFeeder.T_CtrleSingle.lrVelocity:=0.1;
			T_Station.THardware.TAxisToolFeeder.T_CtrleSingle.lrPosition:=0;
			T_Station.THardware.TAxisToolFeeder.T_CtrleSingle.lrDistance:=-2;
			T_Station.THardware.TAxisToolFeeder.T_CtrleSingle.iFunction:=19;
			T_Station.THardware.TAxisToolFeeder.T_CtrleSingle.xExecute:=TRUE;
			(* next step *)
			iStepAction:=30;
			xStepActionDone:=FALSE;
		(* confirm execution *)
		30:	IF NOT(xStepActionDone) THEN
			(* confirm execution *)
				T_Station.THardware.TAxisToolFeeder.T_CtrleSingle.xExecute:=FALSE;
				xStepActionDone:=TRUE;
			ELSE
				IF T_Station.THardware.TAxisToolFeeder.T_CtrleSingle.xDone THEN
					T_Visu.ptrT_ExchgParam^.T_StationCommon.iWireFeederAngleRefIndex:=T_Station.THardware.TAxisToolFeeder.T_CtrleSingle.iStrokeAngleRefIndex;
					xStepActionDone:=FALSE;
					iStepAction:=40;
				ELSE
					IF T_Station.THardware.TAxisToolFeeder.T_CtrleSingle.xErr THEN
					(* activ action not ready or error *)
						iStepAction:=99;
						xStepActionDone:=FALSE;
					END_IF
				END_IF
			END_IF;
		(* Reference axis *)
		40:	T_Station.THardware.TAxisToolFeeder.T_CtrleSingle.lrHomingMethode:=5;
			T_Station.THardware.TAxisToolFeeder.T_CtrleSingle.lrHomeOffset:=0.0;
			T_Station.THardware.TAxisToolFeeder.T_CtrleSingle.lrHomeSpeedSwitch:=T_NovRAM.T_Data.T_Standard.T_TeachINToolFeeder.rRefSpeed;
			T_Station.THardware.TAxisToolFeeder.T_CtrleSingle.lrHomeSpeedZero:=T_NovRAM.T_Data.T_Standard.T_TeachINToolFeeder.rRefSpeed / 10.0;
			T_Station.THardware.TAxisToolFeeder.T_CtrleSingle.lrHomeAcceleration:=T_NovRAM.T_Data.T_Standard.T_TeachINToolFeeder.rAcceleration;
			T_Station.THardware.TAxisToolFeeder.T_CtrleSingle.iFunction:=9;	(* Reference Axis *)
			T_Station.THardware.TAxisToolFeeder.T_CtrleSingle.xExecute:=TRUE;
			(* next step *)
			iStepAction:=50;
			xStepActionDone:=FALSE;
		(* confirm execution *)
		50:	IF NOT(xStepActionDone) THEN
			(* confirm execution *)
				T_Station.THardware.TAxisToolFeeder.T_CtrleSingle.xExecute:=FALSE;
				xStepActionDone:=TRUE;
			ELSE
				IF T_Station.THardware.TAxisToolFeeder.T_CtrleSingle.xDone THEN
				(* confirm action next step *)
					bStateMachine:=1;
					xSetStateMachine:=TRUE;
					iStepAction:=90;
					xStepActionDone:=FALSE;
				ELSE
					IF T_Station.THardware.TAxisToolFeeder.T_CtrleSingle.xErr THEN
					(* activ action not ready or error *)
						iStepAction:=99;
						xStepActionDone:=FALSE;
					END_IF
				END_IF
			END_IF
		(* waiting time out *)
		89:	IF TimerAction.Q THEN iStepAction:=90; END_IF
		(* action done *)
		90:	T_Visu.T_CtrleAction.xDone:=TRUE;
			T_Visu.T_CtrleAction.xNotReady:=FALSE;
			T_Visu.T_CtrleAction.xErr:=FALSE;
			T_Visu.T_CtrleAction.udiErrorID:=0;
			xCalcAngleRefIndex:=FALSE;
		(* axis not ready *)
		95:	TimerNotReady(IN:=TRUE);
			xCalcAngleRefIndex:=FALSE;
		(* error *)
		99:	T_Visu.ptrT_ExchgParam^.T_StationCommon.wState:=T_Visu.ptrT_ExchgParam^.T_StationCommon.wState AND 16#BF;
			T_Visu.T_CtrleAction.xDone:=TRUE;
			T_Visu.T_CtrleAction.xNotReady:=FALSE;
			IF (T_Station.THardware.TAxisToolFeeder.T_Config_Gen.iTyp <> 0) THEN
				diErrorNr:=(T_Station.THardware.TAxisToolFeeder.T_Config_Gen.iTyp * 1000000) + T_Station.THardware.TAxisToolFeeder.T_CtrleSingle.udiErrorID;
			ELSE
				diErrorNr:=0;
			END_IF;
			FBErrorMessage(	diErrorNr:=diErrorNr,
							T_ErrorList:=T_ErrorList);
			T_Visu.ptrT_ExchgParam^.T_Visu.T_Message.sDynamicTextEnglish:=FBErrorMessage.sErrorTextEnglish;
			T_Visu.ptrT_ExchgParam^.T_Visu.T_Message.sDynamicTextDeutsch:=FBErrorMessage.sErrorTextDeutsch;
			T_Visu.ptrT_ExchgParam^.T_Visu.T_Message.sDynamicTextFrancais:=FBErrorMessage.sErrorTextFrancais;
			T_Visu.ptrT_ExchgParam^.T_SafetyCtrl.xSetForceError:=TRUE;
			T_Visu.ptrT_ExchgParam^.T_SafetyCtrl.diSetForceErrorNr:=diErrorNr;
			T_Visu.T_CtrleAction.xErr:=FALSE;
			T_Visu.T_CtrleAction.udiErrorID:=0;
			T_Station.THardware.TAxisToolFeeder.T_CtrleSingle.iFunction:=1;
			T_Station.THardware.TAxisToolFeeder.T_CtrleSingle.xExecute:=TRUE;
			xCalcAngleRefIndex:=FALSE;
		END_CASE
	END_IF;

(* Switch ToolRotation Master Slave *)
	IF xSwitchMasterSlave THEN
		CASE iStepAction OF
		(* check axis *)
		1:	IF NOT T_Station.TControl.xHardwareConfigError THEN
				xStepActionDone:=FALSE;
				iStepAction:=95;
				xTmp:=	T_Station.THardware.TAxisToolLeft.T_CtrleSingle.xDone AND
						T_Station.THardware.TAxisToolLeft.T_CtrleSingle.xNotMoving AND
						NOT(T_Station.THardware.TAxisToolLeft.T_CtrleSingle.xErr) AND
						NOT(T_Station.THardware.TAxisToolLeft.T_CtrleSingle.xExecute);
				xTmp:=	xTmp AND
						((T_Station.THardware.TAxisToolCenter.T_CtrleSingle.xDone AND
						T_Station.THardware.TAxisToolCenter.T_CtrleSingle.xNotMoving AND
						NOT(T_Station.THardware.TAxisToolCenter.T_CtrleSingle.xErr) AND
						NOT(T_Station.THardware.TAxisToolCenter.T_CtrleSingle.xExecute) AND
						xMicroRodActive) OR
						NOT(xMicroRodActive));
				xTmp:=	xTmp AND
						T_Station.THardware.TAxisToolRight.T_CtrleSingle.xDone AND
						T_Station.THardware.TAxisToolRight.T_CtrleSingle.xNotMoving AND
						NOT(T_Station.THardware.TAxisToolRight.T_CtrleSingle.xErr) AND
						NOT(T_Station.THardware.TAxisToolRight.T_CtrleSingle.xExecute);
				xTmp:=	xTmp AND
						((T_Station.THardware.TAxisToolFeeder.T_CtrleSingle.xDone AND
						T_Station.THardware.TAxisToolFeeder.T_CtrleSingle.xNotMoving AND
						NOT(T_Station.THardware.TAxisToolFeeder.T_CtrleSingle.xErr) AND
						NOT(T_Station.THardware.TAxisToolFeeder.T_CtrleSingle.xExecute) AND
						NOT(xMicroRodActive)) OR
						xMicroRodActive);
				(* Start/Stop position or speed of teachin page has to be confirmed *)
				IF xTmp THEN
					iStepAction:=10;
				END_IF
			ELSE
				iStepAction:=95;
			END_IF;
		(* activ function axis *)
		10:	bStateMachine:=2;
			xSetStateMachine:=TRUE;
			T_Station.THardware.TAxisToolRight.T_CtrleSingle.iFunction:=25;
			T_Station.THardware.TAxisToolRight.T_CtrleSingle.xExecute:=TRUE;
			IF xMicroRodActive THEN
				T_Station.THardware.TAxisToolCenter.T_CtrleSingle.iFunction:=25;
				T_Station.THardware.TAxisToolCenter.T_CtrleSingle.xExecute:=TRUE;
			END_IF;
			IF NOT(xMicroRodActive) THEN
				T_Station.THardware.TAxisToolFeeder.T_CtrleSingle.iFunction:=25;
				T_Station.THardware.TAxisToolFeeder.T_CtrleSingle.xExecute:=TRUE;
			END_IF;
			(* next step *)
			iStepAction:=20;
			xStepActionDone:=FALSE;
		(* confirm execution *)
		20:	IF NOT(xStepActionDone) THEN
			(* confirm execution *)
				T_Station.THardware.TAxisToolRight.T_CtrleSingle.xExecute:=FALSE;
				IF xMicroRodActive THEN
					T_Station.THardware.TAxisToolCenter.T_CtrleSingle.xExecute:=FALSE;
				END_IF;
				IF NOT(xMicroRodActive) THEN
					T_Station.THardware.TAxisToolFeeder.T_CtrleSingle.xExecute:=FALSE;
				END_IF;
				xStepActionDone:=TRUE;
			ELSE
				IF T_Station.THardware.TAxisToolRight.T_CtrleSingle.xDone AND ((T_Station.THardware.TAxisToolCenter.T_CtrleSingle.xDone AND xMicroRodActive) OR NOT(xMicroRodActive)) AND
				     ((T_Station.THardware.TAxisToolFeeder.T_CtrleSingle.xDone AND NOT(xMicroRodActive)) OR xMicroRodActive) THEN
				(* confirm action next step *)
					IF T_Station.THardware.TAxisToolRight.T_CtrleSingle.xSlave AND T_Station.THardware.TAxisToolCenter.T_CtrleSingle.xSlave AND xMicroRodActive THEN
						xToolRotationMasterSlave:=TRUE;
					END_IF;
					IF NOT(T_Station.THardware.TAxisToolRight.T_CtrleSingle.xSlave) AND NOT(T_Station.THardware.TAxisToolCenter.T_CtrleSingle.xSlave) AND xMicroRodActive THEN
						xToolRotationMasterSlave:=FALSE;
					END_IF;
					IF T_Station.THardware.TAxisToolRight.T_CtrleSingle.xSlave AND T_Station.THardware.TAxisToolFeeder.T_CtrleSingle.xSlave AND NOT(xMicroRodActive) THEN
						xToolRotationMasterSlave:=TRUE;
					END_IF;
					IF NOT(T_Station.THardware.TAxisToolRight.T_CtrleSingle.xSlave) AND NOT(T_Station.THardware.TAxisToolFeeder.T_CtrleSingle.xSlave) AND NOT(xMicroRodActive) THEN
						xToolRotationMasterSlave:=FALSE;
					END_IF;
					iStepAction:=90;
					xStepActionDone:=FALSE;
				ELSE
					IF T_Station.THardware.TAxisToolRight.T_CtrleSingle.xErr OR (T_Station.THardware.TAxisToolCenter.T_CtrleSingle.xErr AND xMicroRodActive) OR
					     (T_Station.THardware.TAxisToolFeeder.T_CtrleSingle.xErr AND NOT(xMicroRodActive)) THEN
					(* activ action not ready or error *)
						iStepAction:=99;
						xStepActionDone:=FALSE;
					END_IF
				END_IF
			END_IF
		(* action done *)
		90:	bStateMachine:=1;
			xSetStateMachine:=TRUE;
			T_Visu.ptrT_ExchgParam^.T_StationCommon.wState:=T_Visu.ptrT_ExchgParam^.T_StationCommon.wState AND 16#BF;
			T_Visu.T_CtrleAction.xDone:=TRUE;
			T_Visu.T_CtrleAction.xNotReady:=FALSE;
			T_Visu.T_CtrleAction.xErr:=FALSE;
			T_Visu.T_CtrleAction.udiErrorID:=0;
			xSwitchMasterSlave:=FALSE;
		(* axis not ready *)
		95:	T_Visu.ptrT_ExchgParam^.T_StationCommon.wState:=T_Visu.ptrT_ExchgParam^.T_StationCommon.wState AND 16#BF;
			TimerNotReady(IN:=TRUE);
			xSwitchMasterSlave:=FALSE;
		(* error *)
		99:	T_Visu.ptrT_ExchgParam^.T_StationCommon.wState:=T_Visu.ptrT_ExchgParam^.T_StationCommon.wState AND 16#BF;
			T_Visu.T_CtrleAction.xDone:=TRUE;
			T_Visu.T_CtrleAction.xNotReady:=FALSE;
			IF T_Station.THardware.TAxisToolRight.T_CtrleSingle.xErr THEN
				IF (T_Station.THardware.TAxisToolRight.T_Config_Gen.iTyp <> 0) THEN
					diErrorNr:=(T_Station.THardware.TAxisToolRight.T_Config_Gen.iTyp * 1000000) + T_Station.THardware.TAxisToolRight.T_CtrleSingle.udiErrorID;
				ELSE
					diErrorNr:=0;
				END_IF;
			END_IF;
			IF T_Station.THardware.TAxisToolCenter.T_CtrleSingle.xErr AND xMicroRodActive THEN
				IF (T_Station.THardware.TAxisToolCenter.T_Config_Gen.iTyp <> 0) THEN
					diErrorNr:=(T_Station.THardware.TAxisToolCenter.T_Config_Gen.iTyp * 1000000) + T_Station.THardware.TAxisToolCenter.T_CtrleSingle.udiErrorID;
				ELSE
					diErrorNr:=0;
				END_IF;
			END_IF;
			IF T_Station.THardware.TAxisToolFeeder.T_CtrleSingle.xErr AND NOT(xMicroRodActive) THEN
				IF (T_Station.THardware.TAxisToolFeeder.T_Config_Gen.iTyp <> 0) THEN
					diErrorNr:=(T_Station.THardware.TAxisToolFeeder.T_Config_Gen.iTyp * 1000000) + T_Station.THardware.TAxisToolFeeder.T_CtrleSingle.udiErrorID;
				ELSE
					diErrorNr:=0;
				END_IF;
			END_IF;
			FBErrorMessage(	diErrorNr:=diErrorNr,
							T_ErrorList:=T_ErrorList);
			T_Visu.ptrT_ExchgParam^.T_Visu.T_Message.sDynamicTextEnglish:=FBErrorMessage.sErrorTextEnglish;
			T_Visu.ptrT_ExchgParam^.T_Visu.T_Message.sDynamicTextDeutsch:=FBErrorMessage.sErrorTextDeutsch;
			T_Visu.ptrT_ExchgParam^.T_Visu.T_Message.sDynamicTextFrancais:=FBErrorMessage.sErrorTextFrancais;
			T_Visu.ptrT_ExchgParam^.T_SafetyCtrl.xSetForceError:=TRUE;
			T_Visu.ptrT_ExchgParam^.T_SafetyCtrl.diSetForceErrorNr:=diErrorNr;
			T_Visu.T_CtrleAction.xErr:=FALSE;
			T_Visu.T_CtrleAction.udiErrorID:=0;
			T_Station.THardware.TAxisToolRight.T_CtrleSingle.iFunction:=1;
			T_Station.THardware.TAxisToolCenter.T_CtrleSingle.iFunction:=1;
			T_Station.THardware.TAxisToolFeeder.T_CtrleSingle.iFunction:=1;
			T_Station.THardware.TAxisToolRight.T_CtrleSingle.xExecute:=T_Station.THardware.TAxisToolRight.T_CtrleSingle.xErr;
			T_Station.THardware.TAxisToolCenter.T_CtrleSingle.xExecute:=T_Station.THardware.TAxisToolCenter.T_CtrleSingle.xErr AND xMicroRodActive;
			T_Station.THardware.TAxisToolFeeder.T_CtrleSingle.xExecute:=T_Station.THardware.TAxisToolFeeder.T_CtrleSingle.xErr AND NOT(xMicroRodActive);
			xSwitchMasterSlave:=FALSE;
		END_CASE
	END_IF;
END_ACTION
ACTION VisuFunction_Cylinder:
(* Action cylinder toggle state *)
	IF xToggleCylinderState THEN
		(* Step toggle state *)
		CASE iStepAction OF
		(* check cylinder state *)
		1:	xTmp:=	ptrCylAction^.T_CtrleCyl.xDone
					AND NOT(ptrCylAction^.T_CtrleCyl.xExecute)
					AND NOT(ptrCylAction^.T_CtrleCyl.xErr);
			(* next step *)
			IF xTmp THEN iStepAction:=10; ELSE iStepAction:=95; END_IF
			IF xTmp AND T_Station.TControl.xHardwareConfigError THEN iStepAction:=95; END_IF;
		(* toggle cylinder state *)
		10:	ptrCylAction^.T_CtrleCyl.iFunction:=51;
			ptrCylAction^.T_CtrleCyl.xExecute:=TRUE;
			(* next step *)
			iStepAction:=20;
			xStepActionDone:=FALSE;
		(* wait confirmation *)
		20:	IF NOT(xStepActionDone) THEN
			(* release execution *)
				ptrCylAction^.T_CtrleCyl.xExecute:=FALSE;
				xStepActionDone:=TRUE;
			ELSE
				IF ptrCylAction^.T_CtrleCyl.xDone THEN
				(* action done *)
					iStepAction:=90;
					xStepActionDone:=FALSE;
				ELSE 	IF ptrCylAction^.T_CtrleCyl.xErr THEN
						(* action error *)
							iStepAction:=99;
							xStepActionDone:=FALSE;
						END_IF
				END_IF
			END_IF
		(* waiting time out *)
		89:	IF TimerAction.Q THEN iStepAction:=90; END_IF
		(* action done *)
		90:	T_Visu.T_CtrleAction.xDone:=TRUE;
			T_Visu.T_CtrleAction.xNotReady:=FALSE;
			T_Visu.T_CtrleAction.xErr:=FALSE;
			T_Visu.T_CtrleAction.udiErrorID:=0;
			xToggleCylinderState:=FALSE;
		(* cylinder not ready *)
		95:	TimerNotReady(IN:=TRUE);
			xToggleCylinderState:=FALSE;
		(* error *)
		99:	T_Visu.T_CtrleAction.xDone:=TRUE;
			T_Visu.T_CtrleAction.xNotReady:=FALSE;
			(*diErrorNr:=6000000 * ptrCylAction^.T_CtrleCyl.udiErrorID;*)
			diErrorNr:=9000000+ (1000000 * iSelectedCylinder) + ptrCylAction^.T_CtrleCyl.udiErrorID;
			FBErrorMessage(	diErrorNr:=diErrorNr,
							T_ErrorList:=T_ErrorList);
			T_Visu.ptrT_ExchgParam^.T_Visu.T_Message.sDynamicTextEnglish:=FBErrorMessage.sErrorTextEnglish;
			T_Visu.ptrT_ExchgParam^.T_Visu.T_Message.sDynamicTextDeutsch:=FBErrorMessage.sErrorTextDeutsch;
			T_Visu.ptrT_ExchgParam^.T_Visu.T_Message.sDynamicTextFrancais:=FBErrorMessage.sErrorTextFrancais;
			T_Visu.ptrT_ExchgParam^.T_SafetyCtrl.xSetForceError:=TRUE;
			T_Visu.ptrT_ExchgParam^.T_SafetyCtrl.diSetForceErrorNr:=diErrorNr;
			T_Visu.T_CtrleAction.xErr:=FALSE;
			T_Visu.T_CtrleAction.udiErrorID:=0;
			ptrCylAction^.T_CtrleCyl.xReset:=TRUE;
			xToggleCylinderState:=FALSE;
		END_CASE
	END_IF

